// TwinCAT 3 PLC project ExtruderControl
// ProgramVersion: 3.1.4023.0
// libraries:
//   Tc2_ControllerToolbox, * (Beckhoff Automation GmbH)
//   Tc2_MC2, * (Beckhoff Automation GmbH)
//   Tc2_MC2_FlyingSaw, * (Beckhoff Automation GmbH)
//   Tc2_Standard, * (Beckhoff Automation GmbH)
//   Tc2_System, * (Beckhoff Automation GmbH)
//   Tc2_TempController, * (Beckhoff Automation GmbH)
//   Tc3_Database, * (Beckhoff Automation GmbH)
//   Tc3_Module, * (Beckhoff Automation GmbH)
//   VisuDialogs, * (System)
//   VisuSymbols,3.5.10.0,System
// project tree:
//   DUTs/ Modes.TcDUT, ST_CTRL_TempCtrlParameter2.TcDUT, ST_Material.TcDUT
//   DUTs/Vision/ PlcToSensor.TcDUT (not stored), SensorToPlc.TcDUT, VisionCmd.TcDUT, VisionState.TcDUT
//   / GlobalTextList.TcGTLO, PlcTask.TcTTO (not stored), Visualization Manager.TcVMO (not stored)
//   GVLs/ GVL.TcGVL, HMI.TcGVL, IO.TcGVL, MC.TcGVL
//   POUs/ AutoExtrusion.TcPOU (not stored), ControlTemp.TcPOU, GestionVentiladores.TcPOU, MedidaDiamMec.TcPOU, MedidaTempPuente.TcPOU, MAIN.TcPOU, MedidaTempTarjeta.TcPOU, Motion.TcPOU, OperatingModes.TcPOU
//   POUs/Database/ DatabaseManager.TcPOU
//   POUs/Operation/ Basic.TcPOU, Manual.TcPOU
//   POUs/Vision/ SensorFQM.TcPOU
//   POUs/VISUCode/ VisuLogic.TcPOU
//   VISUs/ BasicHMI.TcVIS, MainHMI.TcVIS, ManualHMI.TcVIS, VisionHMI.TcVIS
// real-time tasks:
//   TASK PlcTask: cycle T#10ms, priority 20, ADS port 350
// motion (NC):
//   TASK NC-Task Extruder SAF: cycle T#2ms, priority 4, ADS port 501
//   TASK NC-Task Extruder SVB: cycle T#10ms, priority 8, ADS port 511
//   AXIS ExtruderAxis (id 1)
//     Velo: FastManual=1300
//     PositionAreaControl: Range=50
//     OtherSettings: AllowMotionCmdToSlave=true
//     encoder EncType=8
//       EncPara: ScaleFactorNumerator=360, ScaleFactorDenominator=8388608, Inverse=true, MaxCount=#xffffffff
//     drive DrvType=9
//       DrvPara: Inverse=true, MaxCount=#xffffffff, DriveControlDWord=#x00030000
//         Analog: VeloScale=1.02398817080127, TorqueSetpointScale=10, ScaleFactorActTorque=0.1
//         TimeComp: TaskDelayCycles=1
//     controller CtrType=1
//       CtrPara: PriorControlFactor=1
//         PosDiffControl: Range=50
//         Observer: BandWidth=20
//   AXIS PullerAxis (id 2)
//     General: UnitName=Degree
//     Dynamic: Acceleration=68391, Deceleration=68391, Jerk=205173
//     Velo: RefSearch=455.94, RefSync=455.94, SlowManual=2279.7, FastManual=13678.2, Fast=45594, Maximum=45594
//     OtherSettings: AllowMotionCmdToSlave=true
//     encoder EncType=8
//       EncPara: ScaleFactorNumerator=360, ScaleFactorDenominator=1048576, MaxCount=#xffffffff
//     drive DrvType=9
//       DrvPara: MaxCount=#xffffffff, DriveControlDWord=#x00030000
//         Analog: VeloReferenz=50153.4, VeloScale=1.02398817080127, TorqueSetpointScale=10, ScaleFactorActTorque=0.1
//         TimeComp: TaskDelayCycles=1
//     controller CtrType=1
//       CtrPara: PriorControlFactor=1
//         Observer: BandWidth=20
//   AXIS PullerAxisVirtual (id 3)
//     General: UnitName=Degree
//     OtherSettings: AllowMotionCmdToSlave=true
//     encoder EncType=1
//       EncPara: ScaleFactorNumerator=1
//     drive DrvType=5
//       Analog: TorqueSetpointScale=10, ScaleFactorActTorque=0.1
//       TimeComp: TaskDelayCycles=1
//     controller CtrType=1
//       CtrPara: PriorControlFactor=1
//         Observer: BandWidth=20
// I/O:
//   DEVICE Dispositivo 2 (EtherCAT), AmsNetId 192.168.56.1.3.1
//     Term 1 (EK1100) [EK1100 EtherCAT Coupler (2A E-Bus)]
//       Term 2 (EL2008) [EL2008 8Ch. Dig. Output 24V, 0.5A]
//       Term 6 (EL3102) [EL3102 2Ch. Ana. Input +/-10V, Diff.]
//       Term 8 (EL3102) [EL3102 2Ch. Ana. Input +/-10V, Diff.]
//       Term 11 (EL3202) [EL3202 2Ch. Ana. Input PT100 (RTD)]
//       Term 13 (EL4132) [EL4132 2Ch. Ana. Output +/-10V]
//       Term 15 (EL9011) [EL9011 End Terminal]
//     Drive 3 (AX5206-0000-0011) [AX5206-0000-0011 EtherCAT Drive (SoE, 2 Ch.)]
//     Nº de boxes 7 (FQ-MS12x-ECT) [FQ-MS12x-ECT]
// variable links:
//   NC-Task Extruder SAF/Axes/ExtruderAxis <-> Device 2 (EtherCAT)/Drive 3 (AX5206-0000-0011)
//     Drive/Inputs/In/nDcOutputTime <-> InfoData/DcOutputShift
//     Drive/Inputs/In/nState1 <-> AT 1/Drive status word @bit 8
//     Drive/Inputs/In/nState2 <-> AT 1/Drive status word
//     Drive/Inputs/In/nState4 @bit 1 <-> WcState/InputToggle
//     Drive/Inputs/In/nState4 <-> WcState/WcState
//     Drive/Outputs/Out/nCtrl1 <-> MDT 1/Master control word @bit 8
//     Drive/Outputs/Out/nDataOut2 <-> MDT 1/Velocity command value
//     Enc/Inputs/In/nDataIn1 <-> AT 1/Position feedback 1 value
//     Enc/Inputs/In/nDcInputTime <-> InfoData/DcInputShift
//     Enc/Inputs/In/nState4 @bit 1 <-> WcState/InputToggle
//     Enc/Inputs/In/nState4 <-> WcState/WcState
//   NC-Task Extruder SAF/Axes/PullerAxis <-> Device 2 (EtherCAT)/Drive 3 (AX5206-0000-0011)
//     Drive/Inputs/In/nDcOutputTime <-> InfoData/DcOutputShift
//     Drive/Inputs/In/nState1 <-> AT 2/Drive status word @bit 8
//     Drive/Inputs/In/nState2 <-> AT 2/Drive status word
//     Drive/Inputs/In/nState4 @bit 1 <-> WcState/InputToggle
//     Drive/Inputs/In/nState4 <-> WcState/WcState
//     Drive/Outputs/Out/nCtrl1 <-> MDT 2/Master control word @bit 8
//     Drive/Outputs/Out/nDataOut2 <-> MDT 2/Velocity command value
//     Enc/Inputs/In/nDataIn1 <-> AT 2/Position feedback 1 value
//     Enc/Inputs/In/nDcInputTime <-> InfoData/DcInputShift
//     Enc/Inputs/In/nState4 @bit 1 <-> WcState/InputToggle
//     Enc/Inputs/In/nState4 <-> WcState/WcState
//   ExtruderControl/ExtruderControl Instance <-> Device 2 (EtherCAT)/Nº de boxes 7 (FQ-MS12x-ECT)
//     PlcTask Inputs/GVL.Vision.SensorToPlc/VisionDataOutput <-> 259th transmit PDO Mapping/Vision Data Output1
//     PlcTask Inputs/GVL.Vision.SensorToPlc/VisionDataOutput @bit {32..224 step 32} <-> 259th transmit PDO Mapping/Vision Data Output{2..8}  (7 links)
//     PlcTask Inputs/GVL.Vision.SensorToPlc/VisionResponseCode <-> 258th transmit PDO Mapping/Vision Response Code
//     PlcTask Inputs/GVL.Vision.SensorToPlc/VisionResponseData <-> 258th transmit PDO Mapping/Vision Response Data1
//     PlcTask Inputs/GVL.Vision.SensorToPlc/VisionStatusFlag @bit 1 <-> 257th transmit PDO Mapping/BUSY Bit
//     PlcTask Inputs/GVL.Vision.SensorToPlc/VisionStatusFlag @bit 15 <-> 257th transmit PDO Mapping/ERR Bit
//     PlcTask Inputs/GVL.Vision.SensorToPlc/VisionStatusFlag <-> 257th transmit PDO Mapping/FLG Bit
//     PlcTask Inputs/GVL.Vision.SensorToPlc/VisionStatusFlag @bit 16 <-> 257th transmit PDO Mapping/GATE Bit
//     PlcTask Inputs/GVL.Vision.SensorToPlc/VisionStatusFlag @bit 3 <-> 257th transmit PDO Mapping/OR Bit
//     PlcTask Inputs/GVL.Vision.SensorToPlc/VisionStatusFlag @bit 2 <-> 257th transmit PDO Mapping/READY Bit
//     PlcTask Inputs/GVL.Vision.SensorToPlc/VisionStatusFlag @bit 4 <-> 257th transmit PDO Mapping/RUN Bit
//     PlcTask Inputs/GVL.Vision.SensorToPlc/VisionStatusFlag @bit 5 <-> 257th transmit PDO Mapping/Status Reserve Bit05
//     PlcTask Inputs/GVL.Vision.SensorToPlc/VisionStatusFlag @bit 6 <-> 257th transmit PDO Mapping/Status Reserve Bit06
//     PlcTask Inputs/GVL.Vision.SensorToPlc/VisionStatusFlag @bit 7 <-> 257th transmit PDO Mapping/Status Reserve Bit07
//     PlcTask Inputs/GVL.Vision.SensorToPlc/VisionStatusFlag @bit 8 <-> 257th transmit PDO Mapping/Status Reserve Bit08
//     PlcTask Inputs/GVL.Vision.SensorToPlc/VisionStatusFlag @bit 9 <-> 257th transmit PDO Mapping/Status Reserve Bit09
//     PlcTask Inputs/GVL.Vision.SensorToPlc/VisionStatusFlag @bit 10 <-> 257th transmit PDO Mapping/Status Reserve Bit10
//     PlcTask Inputs/GVL.Vision.SensorToPlc/VisionStatusFlag @bit 11 <-> 257th transmit PDO Mapping/Status Reserve Bit11
//     PlcTask Inputs/GVL.Vision.SensorToPlc/VisionStatusFlag @bit 12 <-> 257th transmit PDO Mapping/Status Reserve Bit12
//     PlcTask Inputs/GVL.Vision.SensorToPlc/VisionStatusFlag @bit 13 <-> 257th transmit PDO Mapping/Status Reserve Bit13
//     PlcTask Inputs/GVL.Vision.SensorToPlc/VisionStatusFlag @bit 14 <-> 257th transmit PDO Mapping/Status Reserve Bit14
//     PlcTask Inputs/GVL.Vision.SensorToPlc/VisionStatusFlag @bit 17 <-> 257th transmit PDO Mapping/Status Reserve Bit17
//     PlcTask Inputs/GVL.Vision.SensorToPlc/VisionStatusFlag @bit 18 <-> 257th transmit PDO Mapping/Status Reserve Bit18
//     PlcTask Inputs/GVL.Vision.SensorToPlc/VisionStatusFlag @bit 19 <-> 257th transmit PDO Mapping/Status Reserve Bit19
//     PlcTask Inputs/GVL.Vision.SensorToPlc/VisionStatusFlag @bit 20 <-> 257th transmit PDO Mapping/Status Reserve Bit20
//     PlcTask Inputs/GVL.Vision.SensorToPlc/VisionStatusFlag @bit 21 <-> 257th transmit PDO Mapping/Status Reserve Bit21
//     PlcTask Inputs/GVL.Vision.SensorToPlc/VisionStatusFlag @bit 22 <-> 257th transmit PDO Mapping/Status Reserve Bit22
//     PlcTask Inputs/GVL.Vision.SensorToPlc/VisionStatusFlag @bit 23 <-> 257th transmit PDO Mapping/Status Reserve Bit23
//     PlcTask Inputs/GVL.Vision.SensorToPlc/VisionStatusFlag @bit 24 <-> 257th transmit PDO Mapping/Status Reserve Bit24
//     PlcTask Inputs/GVL.Vision.SensorToPlc/VisionStatusFlag @bit 25 <-> 257th transmit PDO Mapping/Status Reserve Bit25
//     PlcTask Inputs/GVL.Vision.SensorToPlc/VisionStatusFlag @bit 26 <-> 257th transmit PDO Mapping/Status Reserve Bit26
//     PlcTask Inputs/GVL.Vision.SensorToPlc/VisionStatusFlag @bit 27 <-> 257th transmit PDO Mapping/Status Reserve Bit27
//     PlcTask Inputs/GVL.Vision.SensorToPlc/VisionStatusFlag @bit 28 <-> 257th transmit PDO Mapping/Status Reserve Bit28
//     PlcTask Inputs/GVL.Vision.SensorToPlc/VisionStatusFlag @bit 29 <-> 257th transmit PDO Mapping/Status Reserve Bit29
//     PlcTask Inputs/GVL.Vision.SensorToPlc/VisionStatusFlag @bit 30 <-> 257th transmit PDO Mapping/Status Reserve Bit30
//     PlcTask Inputs/GVL.Vision.SensorToPlc/VisionStatusFlag @bit 31 <-> 257th transmit PDO Mapping/Status Reserve Bit31
//     PlcTask Outputs/GVL.Vision.PlcToSensor/VisionCommand <-> 258th receive PDO Mapping/Vision Command
//     PlcTask Outputs/GVL.Vision.PlcToSensor/VisionControlFlag @bit 2 <-> 257th receive PDO Mapping/Control Reserve Bit02
//     PlcTask Outputs/GVL.Vision.PlcToSensor/VisionControlFlag @bit 3 <-> 257th receive PDO Mapping/Control Reserve Bit03
//     PlcTask Outputs/GVL.Vision.PlcToSensor/VisionControlFlag @bit 4 <-> 257th receive PDO Mapping/Control Reserve Bit04
//     PlcTask Outputs/GVL.Vision.PlcToSensor/VisionControlFlag @bit 5 <-> 257th receive PDO Mapping/Control Reserve Bit05
//     PlcTask Outputs/GVL.Vision.PlcToSensor/VisionControlFlag @bit 6 <-> 257th receive PDO Mapping/Control Reserve Bit06
//     PlcTask Outputs/GVL.Vision.PlcToSensor/VisionControlFlag @bit 7 <-> 257th receive PDO Mapping/Control Reserve Bit07
//     PlcTask Outputs/GVL.Vision.PlcToSensor/VisionControlFlag @bit 8 <-> 257th receive PDO Mapping/Control Reserve Bit08
//     PlcTask Outputs/GVL.Vision.PlcToSensor/VisionControlFlag @bit 9 <-> 257th receive PDO Mapping/Control Reserve Bit09
//     PlcTask Outputs/GVL.Vision.PlcToSensor/VisionControlFlag @bit 10 <-> 257th receive PDO Mapping/Control Reserve Bit10
//     PlcTask Outputs/GVL.Vision.PlcToSensor/VisionControlFlag @bit 11 <-> 257th receive PDO Mapping/Control Reserve Bit11
//     PlcTask Outputs/GVL.Vision.PlcToSensor/VisionControlFlag @bit 12 <-> 257th receive PDO Mapping/Control Reserve Bit12
//     PlcTask Outputs/GVL.Vision.PlcToSensor/VisionControlFlag @bit 13 <-> 257th receive PDO Mapping/Control Reserve Bit13
//     PlcTask Outputs/GVL.Vision.PlcToSensor/VisionControlFlag @bit 14 <-> 257th receive PDO Mapping/Control Reserve Bit14
//     PlcTask Outputs/GVL.Vision.PlcToSensor/VisionControlFlag @bit 17 <-> 257th receive PDO Mapping/Control Reserve Bit17
//     PlcTask Outputs/GVL.Vision.PlcToSensor/VisionControlFlag @bit 18 <-> 257th receive PDO Mapping/Control Reserve Bit18
//     PlcTask Outputs/GVL.Vision.PlcToSensor/VisionControlFlag @bit 19 <-> 257th receive PDO Mapping/Control Reserve Bit19
//     PlcTask Outputs/GVL.Vision.PlcToSensor/VisionControlFlag @bit 20 <-> 257th receive PDO Mapping/Control Reserve Bit20
//     PlcTask Outputs/GVL.Vision.PlcToSensor/VisionControlFlag @bit 21 <-> 257th receive PDO Mapping/Control Reserve Bit21
//     PlcTask Outputs/GVL.Vision.PlcToSensor/VisionControlFlag @bit 22 <-> 257th receive PDO Mapping/Control Reserve Bit22
//     PlcTask Outputs/GVL.Vision.PlcToSensor/VisionControlFlag @bit 23 <-> 257th receive PDO Mapping/Control Reserve Bit23
//     PlcTask Outputs/GVL.Vision.PlcToSensor/VisionControlFlag @bit 24 <-> 257th receive PDO Mapping/Control Reserve Bit24
//     PlcTask Outputs/GVL.Vision.PlcToSensor/VisionControlFlag @bit 25 <-> 257th receive PDO Mapping/Control Reserve Bit25
//     PlcTask Outputs/GVL.Vision.PlcToSensor/VisionControlFlag @bit 26 <-> 257th receive PDO Mapping/Control Reserve Bit26
//     PlcTask Outputs/GVL.Vision.PlcToSensor/VisionControlFlag @bit 27 <-> 257th receive PDO Mapping/Control Reserve Bit27
//     PlcTask Outputs/GVL.Vision.PlcToSensor/VisionControlFlag @bit 28 <-> 257th receive PDO Mapping/Control Reserve Bit28
//     PlcTask Outputs/GVL.Vision.PlcToSensor/VisionControlFlag @bit 29 <-> 257th receive PDO Mapping/Control Reserve Bit29
//     PlcTask Outputs/GVL.Vision.PlcToSensor/VisionControlFlag @bit 30 <-> 257th receive PDO Mapping/Control Reserve Bit30
//     PlcTask Outputs/GVL.Vision.PlcToSensor/VisionControlFlag @bit 31 <-> 257th receive PDO Mapping/Control Reserve Bit31
//     PlcTask Outputs/GVL.Vision.PlcToSensor/VisionControlFlag @bit 16 <-> 257th receive PDO Mapping/DSA Bit
//     PlcTask Outputs/GVL.Vision.PlcToSensor/VisionControlFlag @bit 15 <-> 257th receive PDO Mapping/ERCLR Bit
//     PlcTask Outputs/GVL.Vision.PlcToSensor/VisionControlFlag <-> 257th receive PDO Mapping/EXE Bit
//     PlcTask Outputs/GVL.Vision.PlcToSensor/VisionControlFlag @bit 1 <-> 257th receive PDO Mapping/TRIG Bit
//   ExtruderControl/ExtruderControl Instance <-> Device 2 (EtherCAT)/Term 1 (EK1100)/Term 11 (EL3202)
//     PlcTask Inputs/IO.I_TermB <-> RTD Inputs Channel 2/Value
//     PlcTask Inputs/IO.I_TermT <-> RTD Inputs Channel 1/Value
//   ExtruderControl/ExtruderControl Instance <-> Device 2 (EtherCAT)/Term 1 (EK1100)/Term 13 (EL4132)
//     PlcTask Outputs/IO.Q_Vent1 <-> Channel 1/Output
//     PlcTask Outputs/IO.Q_Vent2 <-> Channel 2/Output
//   ExtruderControl/ExtruderControl Instance <-> Device 2 (EtherCAT)/Term 1 (EK1100)/Term 2 (EL2008)
//     PlcTask Outputs/IO.Q_HeaterB <-> Channel 2/Output
//     PlcTask Outputs/IO.Q_HeaterT <-> Channel 1/Output
//     PlcTask Outputs/IO.Q_VisionLight <-> Channel 3/Output
//   ExtruderControl/ExtruderControl Instance <-> Device 2 (EtherCAT)/Term 1 (EK1100)/Term 6 (EL3102)
//     PlcTask Inputs/IO.I_SMec1 <-> Channel 1/Value
//     PlcTask Inputs/IO.I_SMec2 <-> Channel 2/Value
//   ExtruderControl/ExtruderControl Instance <-> Device 2 (EtherCAT)/Term 1 (EK1100)/Term 8 (EL3102)
//     PlcTask Inputs/IO.I_TermBPuente <-> Channel 2/Value
//     PlcTask Inputs/IO.I_TermTPuente <-> Channel 1/Value
//   ExtruderControl/ExtruderControl Instance <-> NC-Task Extruder SAF/Axes/ExtruderAxis
//     PlcTask Inputs/MC.Extruder.NcToPlc <-> Outputs/ToPlc
//     PlcTask Outputs/MC.Extruder.PlcToNc <-> Inputs/FromPlc
//   ExtruderControl/ExtruderControl Instance <-> NC-Task Extruder SAF/Axes/PullerAxis
//     PlcTask Inputs/MC.Puller.NcToPlc <-> Outputs/ToPlc
//     PlcTask Outputs/MC.Puller.PlcToNc <-> Inputs/FromPlc
//   ExtruderControl/ExtruderControl Instance <-> NC-Task Extruder SAF/Axes/PullerAxisVirtual
//     PlcTask Inputs/MC.PullerVirtual.NcToPlc <-> Outputs/ToPlc
//     PlcTask Outputs/MC.PullerVirtual.PlcToNc <-> Inputs/FromPlc

// ---- DUTs/Modes.TcDUT
{attribute 'qualified_only'}
{attribute 'strict'}
TYPE Modes :
(
	STOP_EM := 0,
	STOP_OP := 1,
	AUTO := 2,
	MAN := 3,
	Stopping := 4
);
END_TYPE

// ---- DUTs/ST_CTRL_TempCtrlParameter2.TcDUT
TYPE ST_CTRL_TempCtrlParameter2 :
STRUCT
  (* general parameters *)
  iMode                     : E_CTRL_ControlMode:=1;
  iReactionOnFailure        : E_CTRL_ReactionOnFailure;
  bSelCtrlParameterSet      : BOOL:=FALSE;
  dwAlarmSupp               : DWORD;
  tCtrlCycleTime            : TIME:=T#100MS;
  tTaskCycleTime            : TIME:=T#10MS;

  (* tuning parameteer *)
  iTuningMode               : E_CTRL_TuneMode:= eCTRL_TuneMode_heating;
  tTuneStabilisation        : TIME       := T#20S;
  fEndTunePercentHeating    : LREAL      := 80.0;
  fYTuneHeating             : LREAL;
  fYStableHeating           : LREAL;
  fEndTunePercentCooling    : LREAL      := 20.0;
  fYTuneCooling             : LREAL;
  fYStableCooling           : LREAL;
  fScalingFactor            : LREAL      := 1.0;

  (* setpoint parameters *)
  fWMin                     : LREAL;
  fWMax                     : LREAL;

  (* start up *)
  bEnableSoftStart          : BOOL;
  bEnableRamping            : BOOL;
  fWStartUp                 : LREAL;
  tStartUp                  : TIME;
  bStartUpRamping           : BOOL;
  fWStartUpVeloPos          : LREAL;
  fWStartUpVeloNeg          : LREAL;
  fWVeloPos                 : LREAL;
  fWVeloNeg                 : LREAL;

  (* actual value parameters *)
  bFilter                   : BOOL;
  tFilter                   : TIME;

  (* deadband parameters *)
  bDeadband                 : BOOL;
  fEDeadband                : LREAL;
  
  (* control value parameters *)
  fYMin                     : LREAL;
  fYMax                     : LREAL;
  fYManual                  : LREAL;
  fYOnFailure               : LREAL;
  tPWMCycleTime             : TIME;
  tPWMMinOffTime            : TIME;
  tPWMMinOnTime             : TIME;
  tPWMWaitingTime           : TIME;
  fYThresholdOff            : LREAL;
  fYThresholdOn             : LREAL;
  nCyclesForSwitchOver      : INT        := 100;

  (* controller settings *)
  bEnablePreController      : BOOL;
  bEnableZones              : BOOL;
  bEnableCVFilter           : BOOL;
  iFilterType               : E_CTRL_FilterType;
  iControllerType           : E_CTRL_ControllerType;

  (* min max temperatures *)
  TempLow                   : LREAL;
  TempLowLow                : LREAL;
  TempHigh                  : LREAL;
  TempHighHigh              : LREAL;
  TempAbsoluteHigh          : LREAL;
  TempAbsoluteLow           : LREAL;

  (* internal tuning parameters *)
  fTuneKp                   : LREAL     := 1.2;
  fTuneTn                   : LREAL     := 2.0;
  fTuneTv                   : LREAL     := 0.42;
  fTuneTd                   : LREAL     := 0.25;
END_STRUCT
END_TYPE

// ---- DUTs/ST_Material.TcDUT
TYPE ST_Material :
STRUCT
	ID: ARRAY[0..15] OF BYTE;
	Name: STRING(50);
	Description: STRING(255);
	BedTemperature: LREAL;
	HotendTemperature: LREAL;
	IdealTempExtr: LREAL;
	MinTempExtr: LREAL;
	MaxTempExtr: LREAL;
END_STRUCT
END_TYPE

// ---- DUTs/Vision/SensorToPlc.TcDUT
TYPE SensorToPlc :
STRUCT
	VisionStatusFlag AT %I*:DWORD; //Doble Palabra que contiene los bits siguientes
	FLG:BOOL; //Posicion 0
	BUSY:BOOL; //Posicion 1
	READY:BOOL; //Posicion 2
	OR_Jud:BOOL; //Posicion 3
	RUN:BOOL; //Posicion 4
	ERR:BOOL; //Posicion 15
	GATE:BOOL; //Posicion 16
	
	VisionResponseCode AT %I*:DWORD;
	VisionResponseData AT %I*:DWORD;
	
	//Lecturas desde el sensor
	VisionDataOutput AT %I*: ARRAY [0..7] OF REAL;
END_STRUCT
END_TYPE

// ---- DUTs/Vision/VisionCmd.TcDUT
{attribute 'qualified_only'}
{attribute 'strict'}
TYPE VisionCmd :
(
	StartSingle := 0,
	StartContinuous := 1,
	StopContinuous := 2,
	ClearValues := 3,
	ClearDataOutputBuffer := 4,
	Reset := 5,
	GetLatestError := 6
);
END_TYPE;

// ---- DUTs/Vision/VisionState.TcDUT
{attribute 'qualified_only'}
{attribute 'strict'}
TYPE VisionState :
(
	Error := 000,
	Checking_error := 001,
	Clear_data := 002,
	Clear_error := 003,
	StandStill := 010,
	Switching_Single := 011,
	Switching_Continuous := 012,
	ContinuousMeasurement := 020,
	Stopping_Continuous := 021,
	SingleMeasurement := 030,
	TakingSingleMeasurement := 031,
	EmptyDebug := 999
);
END_TYPE

// ---- GVLs/GVL.TcGVL
{attribute 'qualified_only'}
VAR_GLOBAL
	
	Mode: Modes;
	Vision:SensorFQM;
	VisionResults:ARRAY [0..7] OF REAL;
	VisionResultsmm:ARRAY [0..7] OF REAL;
	//ScalingFactor:REAL:= 0.0414;
	ScalingFactor:REAL:= 0.03798; 	//Factor de escalado (mm/pixeles) para broca de 1.75mm
	
	NuevaMedidaCamara:BOOL:=FALSE; 	//Variable auxiliar para el control de la camara
	
	//Variables para el control de la temperatura
	TempTerT: LREAL; 	//Temperatura medida por el Pt100 del termico superior
	TempTerB: LREAL; 	//Temperatura medida por el Pt100 del termico inferior
	//TempExtrusion:REAL:=205;	//Temperatura de extrusion dependiendo del material (PLA)
	TempExtrusion:REAL:=195;	//Para pruebas
	
	//Variables para el control del diametro del filamento con el sensor mecanico
	MedidaSensorMecanico:REAL:=0.0;		//Media de medidas y por tanto medida del diametro
	
	//Variables para el control del diametro
	config:BOOL:=0; 			//0 para 1.75mm y 1 para 2.85mm de diametro
	dReferencia:REAL:=1.75; 	//1.75 o 2.85
	//Estos valores (vPaso y dTolerancia) habría que asignarlos de forma correcta segun los parametros del motor inferior
	vPaso:INT:=2; 				//Valor para variar la velocidad de actuacion de los rodillos inferiores
	dTolerancia:REAL:=0.03; 	//Tolerancia permitida en la medida del diametro del filamento
	
	//Variable para controlar velocidad del motor inferior (puller)
	//A estas variables habria que asignarle unos valores correctos para realizar el control de forma optima
	ActPuller: LREAL; 			//Valor inicial de actuacion que variara segun el valor del diametro
	ActPuller_Max: LREAL;
	ActPuller_Min: LREAL;
	
	State:INT:= 0; //Para gestion de la maquina de estados
	//0: estado inicial
	//1: dar potencia
	//2: calentar 
	//3: mover en velocidad extrusora y puller
	//4: funcionamiento extrusora
	//5: nueva foto y gestion de termicos
	//6: calculo de la nueva velocidad
	//7: cambio de velocidad del puller
	//30: parar ejes
END_VAR

// ---- GVLs/HMI.TcGVL
{attribute 'qualified_only'}
VAR_GLOBAL
	
	// Modes control
	Bt_Run: BOOL;
	Bt_Stop: BOOL;
	S_ManAuto: BOOL := TRUE;
	Bt_EmStop: BOOL;
	Bt_Rearm:BOOL;
	Bt_Front: BOOL;
	Bt_Back:BOOL;
	
	//Process Control
	Bt_StartCycle:BOOL;
	Bt_StopCycle:BOOL;
	Bt_ResetAxis:BOOL;
	Tb_Vel:LREAL;
	Tb_TempB:LREAL;
	Tb_TempT:LREAL;
	Tb_Temp:LREAL;
	
	//Vision control
	Bt_ActivateContinuous:BOOL;
	Bt_ActivateSingle:BOOL;
	Bt_Shot:BOOL;
	L_NewMeasurement:BOOL;
	
	//Manual HMI
	Bt_ManHeatTop:BOOL;
	Bt_ManHeatBot:BOOL;
	Bt_ManForwardExtruder:BOOL;
	Bt_ManBackwardsExtruder:BOOL;
	Bt_Light:BOOL;
	Tb_ManVelExtruder:REAL;
	Bt_ManForwardPuller:BOOL;
	Bt_ManBackwardsPuller:BOOL;
	Tb_ManVelPuller:REAL;
	
END_VAR

VAR_GLOBAL CONSTANT
	MeasurementNames: ARRAY [0..7] OF STRING:= ['Top diameter','Mid diameter','Low diameter','Empty','Empty','Empty','Empty','Empty'];
END_VAR

// ---- GVLs/IO.TcGVL
{attribute 'qualified_only'}
VAR_GLOBAL
	
	// Heater outputs
	Q_HeaterT AT %Q*:BOOL;
	Q_HeaterB AT %Q*:BOOL;
	Q_VisionLight AT %Q*:BOOL;
	
	// RTD Sensors (PT100)
	I_TermT AT %I*:INT;
	I_TermB AT %I*:INT;
	
	// Valor temperatura puente de resistencias
	I_TermTPuente AT %I*:INT;
	I_TermBPuente AT %I*:INT;
	
	// Sensores mecanicos diametro
	I_SMec1 AT %I*:INT;
	I_SMec2 AT %I*:INT;
	
	//Ventiladores
	Q_Vent1 AT %Q*:INT;
	Q_Vent2 AT %Q*:INT;
	
END_VAR

// ---- GVLs/MC.TcGVL
{attribute 'qualified_only'}
VAR_GLOBAL
	// Axis ref
	Extruder: AXIS_REF;
	Puller: AXIS_REF;
	PullerVirtual:AXIS_REF; //Eje virtual para controlar el Puller
	
	// Orders
	En_Power:BOOL;
	Exec_Stop:BOOL;
	Exec_Velocity:BOOL;
	Exec_Relative:BOOL;
	Exec_Reset:BOOL;
	
	Man_ForwardExtruder:BOOL;
	Man_BackwardsExtruder:BOOL;
	
	Man_ForwardPuller:BOOL;
	Man_BackwardsPuller:BOOL;
	
	// Motion variables
	Override:LREAL := 100;
	TargetVel:LREAL;
	TargetPosRel:LREAL;
	TargetDirection:MC_Direction;
	
	// Puller
	PullerVel:LREAL;
	Exec_VelocityPuller:BOOL;
	PullerDirection:MC_Direction;
	Acoplar:BOOL;
	Desacoplar:BOOL;
END_VAR

VAR_GLOBAL CONSTANT
	// Motion constants
	StdVel:LREAL:= 100;
	StdAcc:LREAL:= 1000;
	StdDecc:LREAL:= 1000;
END_VAR

// ---- POUs/Vision/SensorFQM.TcPOU
FUNCTION_BLOCK SensorFQM
VAR_INPUT
END_VAR
VAR_OUTPUT
END_VAR
VAR_IN_OUT
	
END_VAR
VAR
	State:VisionState:= 0;
	SensorToPlc AT %I*:SensorToPlc;
	PlcToSensor AT %Q*:PlcToSensor;
	KeepAliveTimer:TON;
	
	RExec:R_TRIG;
	NextCycleResetFlags:BOOL;
	Results: ARRAY [0..7] OF REAL;
	
	//Single measurement
	RequestSingle:BOOL;
	TakePhoto:BOOL;
	TakePhotoFlag:R_TRIG;
	MeasureTimer:TON;
	MeasureTime:TIME;
	
	//Continuous measurement
	RequestStartCont:BOOL;
	RequestStopCont:BOOL;
	StopFromError:BOOL;
	ResponseTimer:TON;
	ResponseTime:TIME;
	FEnable:F_TRIG;
	
	LastResult:INT:=0;//0-Null, 1-Ok, 2-NG
	
	//Error Management
	RequestErrorCode:BOOL;
	LastError:DWORD;
END_VAR
VAR CONSTANT
	KeepAliveBit:INT:=24;
END_VAR

// Preparing Inputs
SensorToPlc.FLG:= SensorToPlc.VisionStatusFlag.0;
SensorToPlc.BUSY:= SensorToPlc.VisionStatusFlag.1;
SensorToPlc.READY:= SensorToPlc.VisionStatusFlag.2;
SensorToPlc.OR_Jud:= SensorToPlc.VisionStatusFlag.3;
SensorToPlc.RUN:= SensorToPlc.VisionStatusFlag.4;
SensorToPlc.ERR:= SensorToPlc.VisionStatusFlag.15;
SensorToPlc.GATE:= SensorToPlc.VisionStatusFlag.16;
//Change a bit every 500ms as Keep Alive bit
(*KeepAliveTimer(in:=NOT KeepAliveTimer.Q, pt:=T#1S);
IF KeepAliveTimer.Q THEN
	PlcToSensor.VisionControlFlag.24:= NOT PlcToSensor.VisionControlFlag.24;
END_IF*)

//Delete variables. Estado distinto de 999 para permitir modificar a mano en ese estado especial
IF State <> 999 THEN
	PlcToSensor.EXE:=FALSE;
	PlcToSensor.ERCLR:=FALSE;
	PlcToSensor.DSA:=FALSE;
	PlcToSensor.TRIG:=FALSE;
END_IF

//State machine
CASE State OF
	000: //Error. Por ahora se salta parada cuando hay error
		IF NOT SensorToPlc.ERR THEN
			State := 010;
		ELSE
			State := 001;
		END_IF
			
	001: //Checking errors
		//TODO: Revisar
		_prepareCommand(Command:= VisionCmd.GetLatestError);
		PlcToSensor.EXE := TRUE;
		IF SensorToPlc.FLG THEN
			PlcToSensor.EXE := FALSE;
			LastError:= SensorToPlc.VisionResponseData;
			State := 002;
		END_IF
	002: //Clear data
		_prepareCommand(VisionCmd.ClearDataOutputBuffer);
		PlcToSensor.EXE := TRUE;
		IF SensorToPlc.FLG THEN
			PlcToSensor.EXE := FALSE;
			State := 003;
		END_IF
	003: //Clear Error
		PlcToSensor.ERCLR:=TRUE;
		IF NOT SensorToPlc.ERR THEN
			PlcToSensor.ERCLR := FALSE;
			State := 010;
		END_IF
	010: //StandStill
		IF RequestSingle THEN
			LastError := 0; //Elimina ultimo error cuando se pasa a este estado
			State := 011;
		END_IF
		IF RequestStartCont AND NOT RequestSingle THEN
			State := 012;
		END_IF
		IF SensorToPlc.ERR THEN
			State := 001;
			
		END_IF
	011: //Switching to Single
		_prepareCommand(VisionCmd.StartSingle);
		PlcToSensor.EXE:=TRUE;
		IF SensorToPlc.FLG THEN
			PlcToSensor.EXE := FALSE;
			State := 030;
			LastResult:=0;
		END_IF
	012: //Switching to continuous
		_prepareCommand(VisionCmd.StartContinuous);
		PlcToSensor.EXE:=TRUE;
		IF SensorToPlc.FLG THEN
			PlcToSensor.EXE := FALSE;
			State := 020;
		END_IF
	020: //Continuous Measurement
		//Loop to request measurement
		IF SensorToPlc.GATE THEN
			ResponseTime:=ResponseTimer.ET;
			PlcToSensor.DSA := FALSE;
			ResponseTimer(in:=FALSE, pt:=T#10S);
		ELSIF NOT SensorToPLC.gate THEN
			ResponseTimer(in:=TRUE, pt:=T#10S);
			PlcToSensor.DSA := TRUE;
		END_IF
		//transitions
		IF SensorToPLC.ERR THEN
			PlcToSensor.EXE := FALSE;
			StopFromError:=TRUE;
			State := 021;
		END_IF 
		IF RequestStopCont THEN
			PlcToSensor.EXE := FALSE;
			State := 021;
		END_IF
	021: //Stopping continuous
	    _prepareCommand(VisionCmd.StopContinuous);
		PlcToSensor.EXE := TRUE;
		IF SensorToPLC.FLG THEN
			IF StopFromError THEN
				PlcToSensor.EXE :=FALSE;
				StopFromError:=FALSE;
				State := 001;
			ELSE
				State := 010;
			END_IF
			RequestStopCont := FALSE;
		END_IF
	030: // Single Measurement Ready
		
		IF TakePhoto THEN
			//Take photo and request
			PlcToSensor.TRIG:=TRUE;
			PlcToSensor.DSA:=TRUE;
			MeasureTimer(in:=FALSE);
			MeasureTimer(in:=TRUE, pt:=T#60s);
			State := 31;
		END_IF
		IF NOT RequestSingle THEN
			State := 010;
		END_IF
		IF SensorToPlc.ERR THEN
			State := 001;
			_prepareCommand(Command:= VisionCmd.GetLatestError);
			PlcToSensor.EXE := TRUE;
		END_IF
	031: // Single Measurement Taking photo
		PlcToSensor.DSA := TRUE; // Ojo, ya se activo en el ciclo anterior. no hay retardo de un ciclo.
		PlcToSensor.TRIG := TRUE;
		MeasureTimer(in:=TRUE);
		IF SensorToPLC.GATE THEN
			//TODO: Esto llega mas tarde que el dato. Revisar.
			IF SensorToPlc.OR_Jud THEN
				LastResult:=2;
			ELSE
				LastResult:=1;
			END_IF
			MeasureTime:=MeasureTimer.ET;
			MeasureTimer(in:=FALSE);
			State := 030;
			PlcToSensor.TRIG:=FALSE;
			PlcToSensor.DSA:=FALSE;
		END_IF
		IF SensorToPLC.ERR THEN
			State := 001;
		END_IF
END_CASE

//Update Flag Bits into DWORD
PlcToSensor.VisionControlFlag.0:= PlcToSensor.EXE;
PlcToSensor.VisionControlFlag.1:= PlcToSensor.TRIG;
PlcToSensor.VisionControlFlag.15:= PlcToSensor.ERCLR;
PlcToSensor.VisionControlFlag.16:= PlcToSensor.DSA;

METHOD PRIVATE _prepareCommand
VAR_INPUT
	Command:VisionCmd;
END_VAR
VAR
	
END_VAR
(* 
Command orders deliverable to camera.
See OMRON FQ-M Series Vision Sensor docs for information
*)
CASE Command OF
	VisionCmd.StartSingle: 				PlcToSensor.VisionCommand:= 16#00101010;
	VisionCmd.StartContinuous: 			PlcToSensor.VisionCommand:= 16#00101020;
	VisionCmd.StopContinuous: 			PlcToSensor.VisionCommand:= 16#00101030;
	VisionCmd.ClearValues: 				PlcToSensor.VisionCommand:= 16#00102010;
	VisionCmd.ClearDataOutputBuffer: 	PlcToSensor.VisionCommand:= 16#00102020;
	VisionCmd.Reset: 					PlcToSensor.VisionCommand:= 16#0010F010;
	VisionCmd.GetLatestError: 			PlcToSensor.VisionCommand:= 16#00205000;
END_CASE
END_METHOD

METHOD PUBLIC ContinuousShot : BOOL
VAR_INPUT
	Enable:BOOL; //Habilita el modo continuo. NOTA: Tendrá prioridad el modo único
END_VAR
VAR_OUTPUT
	Q:ARRAY [0..7] OF REAL;
END_VAR
FEnable(CLK:=Enable);
IF Enable THEN
	RequestStartCont:=TRUE;
	RequestStopCont:=FALSE;
END_IF
IF FEnable.Q THEN
	RequestStartCont:=FALSE;
	RequestStopCont:=TRUE;
	PlcToSensor.DSA:=FALSE;
	ResponseTimer(in:=FALSE);
END_IF

IF Enable THEN
//	IF SensorToPlc.GATE THEN
//		ResponseTime:=ResponseTimer.ET;
//		PlcToSensor.DSA := FALSE;
//		ResponseTimer(in:=FALSE, pt:=T#10S);
//	ELSIF NOT SensorToPLC.gate THEN
//		ResponseTimer(in:=TRUE, pt:=T#10S);
//		PlcToSensor.DSA := TRUE;
//	END_IF
;
END_IF

Q := SensorToPlc.VisionDataOutput;
END_METHOD

METHOD PUBLIC SingleShot : BOOL
VAR_INPUT
	Enable:BOOL;
	Execute:BOOL;
END_VAR
VAR_OUTPUT
	Active:BOOL;
	Measurement:BOOL;
	Ok:BOOL;
	Ng:BOOL;
	Q: ARRAY [0..7] OF REAL;
END_VAR
IF Enable THEN
	RequestSingle:=TRUE;
ELSE
	RequestSingle:=FALSE;
END_IF

TakePhotoFlag(clk:= Execute);
IF State = 030 THEN
	Active:=TRUE;
	IF TakePhotoFlag.Q THEN
		TakePhoto:=TRUE;
		Ok:=FALSE;
		Ng:=FALSE;
	END_IF
	CASE LastResult OF
		0: Ok:=FALSE; Ng:=FALSE; Measurement:=FALSE;
		1: Ok:=TRUE; Ng:=FALSE; Measurement:=TRUE;
		2: Ok:=FALSE; Ng:=TRUE; Measurement:= TRUE;
	END_CASE
	
ELSIF State = 031 THEN
	TakePhoto:=FALSE;
END_IF

Q := SensorToPlc.VisionDataOutput;
END_METHOD

END_FUNCTION_BLOCK

// ---- POUs/Operation/Manual.TcPOU
PROGRAM Manual
VAR
	
	ExitManual:F_TRIG;
	
	LoopCounter:INT;
	
	//Variables para la lectura de sensores
	MedSensores:REAL:=0.0;
	SumSenOpt: REAL:=0.0;
	MedSenOpt: REAL:=0.0;
	
	//Variables para la media de medidas de los sensores
	Lecturas:ARRAY[0..9] OF REAL:=[10(0.0)]; 	//Medidas del diametro inicializadas
	Index:INT:=0; 								//Indice del vector de medidas 
	Suma:REAL:=0.0; 							//Suma de medidas
	Medida:REAL:=0.0; 							//Media de medidas y por tanto medida del diametro
	
END_VAR

IF GVL.Mode = Modes.MAN THEN
	//Gestion de temperatura para extrusion.
	//IO.Q_HeaterB:=HMI.Bt_ManHeatBot;
	//IO.Q_HeaterT:=HMI.Bt_ManHeatTop;
	
	IF (GVL.TempTerT>(GVL.TempExtrusion*0.95)) OR (NOT HMI.Bt_ManHeatTop) THEN 	//Gestiona el calentador superior
		IO.Q_HeaterT:=FALSE;
	END_IF
	IF (GVL.TempTerT<(GVL.TempExtrusion*0.95-1.0)) AND HMI.Bt_ManHeatTop THEN
		IO.Q_HeaterT:=TRUE;
	END_IF
	
	IF (GVL.TempTerB>(GVL.TempExtrusion)) OR (NOT HMI.Bt_ManHeatBot) THEN 		//Gestiona el calentador inferior
		IO.Q_HeaterB:=FALSE;
	END_IF
	IF (GVL.TempTerB<(GVL.TempExtrusion-1.0))AND HMI.Bt_ManHeatBot THEN
		IO.Q_HeaterB:=TRUE;
	END_IF
	
	//Al pulsar botones, primero dar orden de potencia
	IF HMI.Bt_ManForwardExtruder OR HMI.Bt_ManBackwardsExtruder OR HMI.Bt_ManBackwardsPuller OR HMI.Bt_ManForwardPuller THEN
		MC.En_Power := TRUE;
		//Ya en potencia, se ejecuta la orden
		IF Motion.FB_Power.Status AND Motion.FB_Power2.Status AND Motion.FB_Power3.Status THEN
			MC.Man_ForwardExtruder := HMI.Bt_ManForwardExtruder;
			MC.Man_BackwardsExtruder := HMI.Bt_ManBackwardsExtruder;
			MC.Man_ForwardPuller:=HMI.Bt_ManForwardPuller;
			MC.Man_BackwardsPuller:=HMI.Bt_ManBackwardsPuller;
		END_IF
	//Si se deja de pulsar, al acabar movimiento, se quita potencia
	ELSE
		MC.Man_ForwardExtruder := FALSE;
		MC.Man_BackwardsExtruder := FALSE;
		MC.Man_ForwardPuller:=FALSE;
		MC.Man_BackwardsPuller:=FALSE;
		IF NOT Motion.FB_ManualExtruder.Busy AND NOT Motion.FB_ManualPuller.Busy THEN
			MC.En_Power := FALSE;
		ELSE
			MC.En_Power := TRUE;
		END_IF
	END_IF
//	MC.Man_Forward := HMI.Bt_ManForward;
//	MC.Man_Backwards := HMI.Bt_ManBackwards;
	IO.Q_VisionLight := HMI.Bt_Light;
	
	GVL.Vision.SingleShot(Enable:=HMI.Bt_ActivateSingle, 
						Execute:=HMI.Bt_Shot,
						Q=>GVL.VisionResults,
						Measurement=>GVL.NuevaMedidaCamara);
    GVL.Vision.ContinuousShot(Enable:=HMI.Bt_ActivateContinuous,
						Q=>GVL.VisionResults);		
	
	IF HMI.Bt_ActivateSingle AND GVL.NuevaMedidaCamara THEN
		// Restablecer valores de medida para una futura medida
		GVL.NuevaMedidaCamara:=FALSE;
		GVL.Vision.SingleShot(Enable:=TRUE, Execute:=FALSE);
		SumSenOpt:=0.0;
		FOR LoopCounter:=0 TO 7 BY 1 DO
			GVL.VisionResultsmm[LoopCounter] := GVL.VisionResults[LoopCounter]*GVL.ScalingFactor;
			SumSenOpt:=GVL.VisionResultsmm[LoopCounter]+SumSenOpt;
		END_FOR	
		MedSenOpt:=SumSenOpt/3;
		
		//Calculo del diametro
		MedSensores:=((GVL.MedidaSensorMecanico+MedSenOpt)/2);
		(*
		//Hacer media de las 10 ultimas medidas del diametro
		Suma:= Suma - Lecturas[Index];
		Lecturas[index]:=MedSensores;
		Suma:=Suma+Lecturas[index];
		Index:= Index + 1;
		IF (Index > 9) THEN
			Index := 0;    	//Volvemos al inicio del vector
		END_IF
		Medida:=Suma/10;
		*)
		(*
		//Gestion de la actuacion
		IF (MedSensores>(GVL.dReferencia+GVL.dTolerancia)) THEN 		//Diametro grande
			GVL.ActPuller:=GVL.ActPuller+GVL.vPaso;
		END_IF
	
		IF (MedSensores<(GVL.dReferencia-GVL.dTolerancia)) THEN 		//Diametro pequeño
			GVL.ActPuller:=GVL.ActPuller-GVL.vPaso;
		END_IF
	
		//Limitador de la actuacion
		IF (GVL.ActPuller>GVL.ActPuller_Max) THEN 
			GVL.ActPuller:=GVL.ActPuller_Max;
		ELSIF (GVL.ActPuller<GVL.ActPuller_Min) THEN
			GVL.ActPuller:=GVL.ActPuller_Min;
		END_IF
		*)
	END_IF
	IF HMI.Bt_ActivateContinuous THEN
		// Restablecer valores de medida para una futura medida
		SumSenOpt:=0.0;
		FOR LoopCounter:=0 TO 7 BY 1 DO
			GVL.VisionResultsmm[LoopCounter] := GVL.VisionResults[LoopCounter]*GVL.ScalingFactor;
			SumSenOpt:=GVL.VisionResultsmm[LoopCounter]+SumSenOpt;
		END_FOR	
		MedSenOpt:=SumSenOpt/3;
		
		//Calculo del diametro
		MedSensores:=((GVL.MedidaSensorMecanico+MedSenOpt)/2);
		
		//Hacer media de las 10 ultimas medidas del diametro
		Suma:= Suma - Lecturas[Index];
		Lecturas[index]:=MedSensores;
		Suma:=Suma+Lecturas[index];
		Index:= Index + 1;
		IF (Index > 9) THEN
			Index := 0;    	//Volvemos al inicio del vector
		END_IF
		Medida:=Suma/10;
		(*
		//Gestion de la actuacion
		IF (MedSensores>(GVL.dReferencia+GVL.dTolerancia)) THEN 		//Diametro grande
			GVL.ActPuller:=GVL.ActPuller+GVL.vPaso;
		END_IF
	
		IF (MedSensores<(GVL.dReferencia-GVL.dTolerancia)) THEN 		//Diametro pequeño
			GVL.ActPuller:=GVL.ActPuller-GVL.vPaso;
		END_IF
	
		//Limitador de la actuacion
		IF (GVL.ActPuller>GVL.ActPuller_Max) THEN 
			GVL.ActPuller:=GVL.ActPuller_Max;
		ELSIF (GVL.ActPuller<GVL.ActPuller_Min) THEN
			GVL.ActPuller:=GVL.ActPuller_Min;
		END_IF
		*)
	END_IF
	
ELSE
	HMI.Bt_ManHeatBot := FALSE;
	HMI.Bt_ManHeatTop:= FALSE;
	MC.Man_ForwardExtruder := FALSE;
	HMI.Bt_ManForwardExtruder := FALSE;
	MC.Man_BackwardsExtruder := FALSE;
	HMI.Bt_ManBackwardsExtruder := FALSE;
	MC.Man_ForwardPuller := FALSE;
	HMI.Bt_ManForwardPuller := FALSE;
	MC.Man_BackwardsPuller := FALSE;
	HMI.Bt_ManBackwardsPuller := FALSE;
	HMI.Bt_Light := FALSE;
	HMI.Bt_ActivateSingle:=FALSE;
	HMI.Bt_ActivateContinuous:=FALSE;
END_IF

ExitManual(clk:=(GVL.Mode = Modes.MAN));
IF ExitManual.Q THEN
	IO.Q_HeaterB := FALSE;
	IO.Q_HeaterT :=FALSE;
	IO.Q_VisionLight := FALSE;
END_IF

END_PROGRAM

// ---- POUs/Motion.TcPOU
PROGRAM Motion
VAR
	FB_Power: MC_Power;
	FB_Stop: MC_Stop;
	FB_StopPuller: MC_Stop;
	FB_StopPullerVirtual: MC_Stop;
	FB_Velocity: MC_MoveVelocity;
	FB_VelocityPuller: MC_MoveVelocity;
	FB_Relative: MC_MoveRelative;
	FB_ReadStatusExtruder: MC_ReadStatus;
	FB_ReadStatusPuller: MC_ReadStatus;
	FB_ResetExtruder: MC_Reset;
	FB_ResetPuller: MC_Reset;
	FB_ManualExtruder: MC_Jog;
	FB_ManualPuller: MC_Jog;
	FB_Power2: MC_Power;
	FB_Power3: MC_Power;
	FB_GearInVelo: MC_GearInVelo;
	FB_GearOut: MC_GearOut;
END_VAR

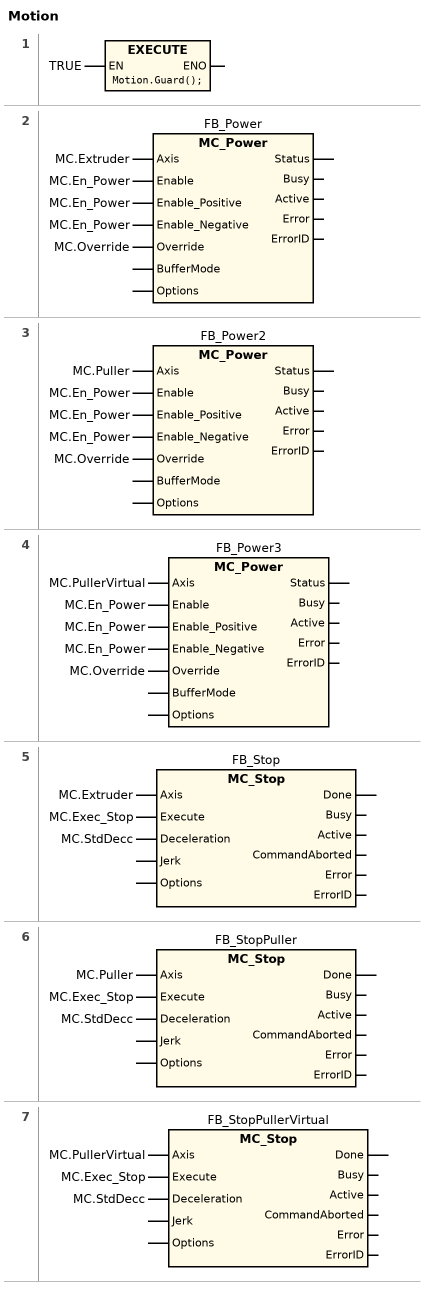
// NETWORK 1
Motion.Guard();

// NETWORK 2
FB_Power(
    Axis := MC.Extruder,
    Enable := MC.En_Power,
    Enable_Positive := MC.En_Power,
    Enable_Negative := MC.En_Power,
    Override := MC.Override); // MC_Power

// NETWORK 3
FB_Power2(
    Axis := MC.Puller,
    Enable := MC.En_Power,
    Enable_Positive := MC.En_Power,
    Enable_Negative := MC.En_Power,
    Override := MC.Override); // MC_Power

// NETWORK 4
FB_Power3(
    Axis := MC.PullerVirtual,
    Enable := MC.En_Power,
    Enable_Positive := MC.En_Power,
    Enable_Negative := MC.En_Power,
    Override := MC.Override); // MC_Power

// NETWORK 5
FB_Stop(Axis := MC.Extruder, Execute := MC.Exec_Stop, Deceleration := MC.StdDecc); // MC_Stop

// NETWORK 6
FB_StopPuller(Axis := MC.Puller, Execute := MC.Exec_Stop, Deceleration := MC.StdDecc); // MC_Stop

// NETWORK 7
FB_StopPullerVirtual(Axis := MC.PullerVirtual, Execute := MC.Exec_Stop, Deceleration := MC.StdDecc); // MC_Stop

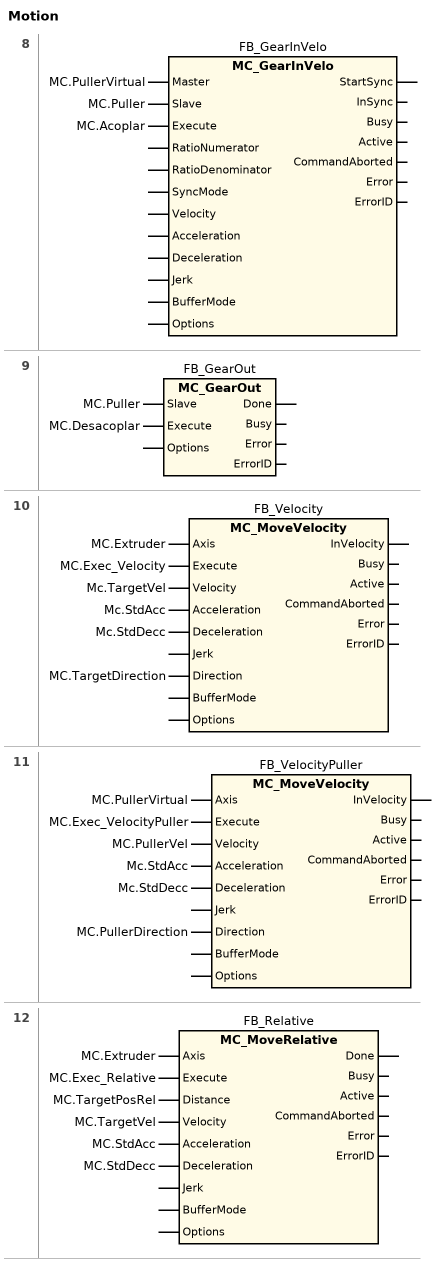
// NETWORK 8
FB_GearInVelo(Master := MC.PullerVirtual, Slave := MC.Puller, Execute := MC.Acoplar); // MC_GearInVelo

// NETWORK 9
FB_GearOut(Slave := MC.Puller, Execute := MC.Desacoplar); // MC_GearOut

// NETWORK 10
FB_Velocity(
    Axis := MC.Extruder,
    Execute := MC.Exec_Velocity,
    Velocity := Mc.TargetVel,
    Acceleration := Mc.StdAcc,
    Deceleration := Mc.StdDecc,
    Direction := MC.TargetDirection); // MC_MoveVelocity

// NETWORK 11
FB_VelocityPuller(
    Axis := MC.PullerVirtual,
    Execute := MC.Exec_VelocityPuller,
    Velocity := MC.PullerVel,
    Acceleration := Mc.StdAcc,
    Deceleration := Mc.StdDecc,
    Direction := MC.PullerDirection); // MC_MoveVelocity

// NETWORK 12
FB_Relative(
    Axis := MC.Extruder,
    Execute := MC.Exec_Relative,
    Distance := MC.TargetPosRel,
    Velocity := MC.TargetVel,
    Acceleration := MC.StdAcc,
    Deceleration := MC.StdDecc); // MC_MoveRelative

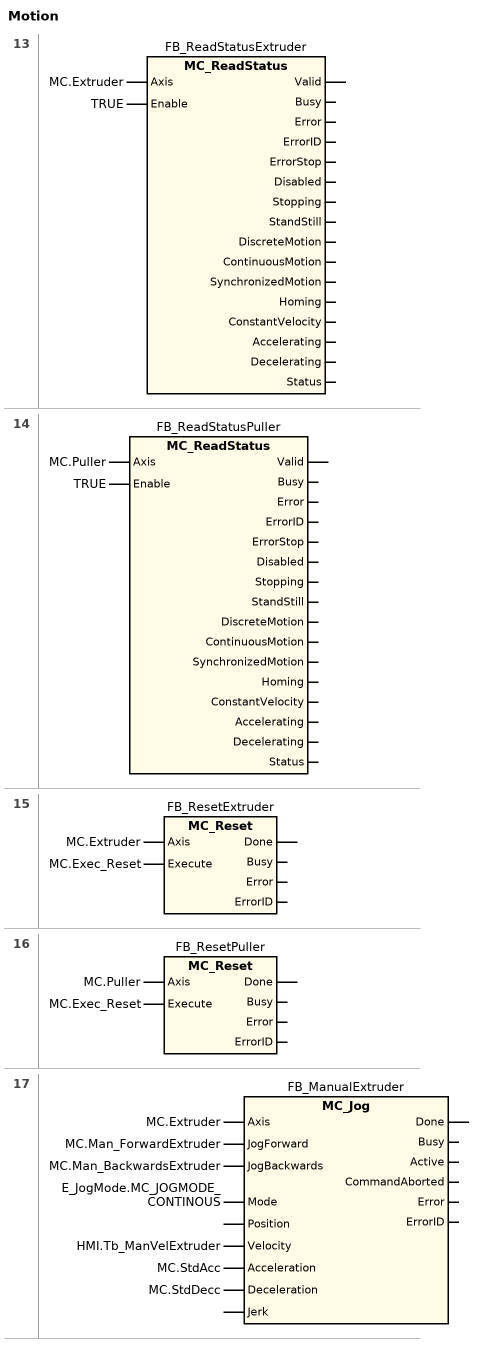
// NETWORK 13
FB_ReadStatusExtruder(Axis := MC.Extruder, Enable := TRUE); // MC_ReadStatus

// NETWORK 14
FB_ReadStatusPuller(Axis := MC.Puller, Enable := TRUE); // MC_ReadStatus

// NETWORK 15
FB_ResetExtruder(Axis := MC.Extruder, Execute := MC.Exec_Reset); // MC_Reset

// NETWORK 16
FB_ResetPuller(Axis := MC.Puller, Execute := MC.Exec_Reset); // MC_Reset

// NETWORK 17
FB_ManualExtruder(
    Axis := MC.Extruder,
    JogForward := MC.Man_ForwardExtruder,
    JogBackwards := MC.Man_BackwardsExtruder,
    Mode := E_JogMode.MC_JOGMODE_CONTINOUS,
    Velocity := HMI.Tb_ManVelExtruder,
    Acceleration := MC.StdAcc,
    Deceleration := MC.StdDecc); // MC_Jog

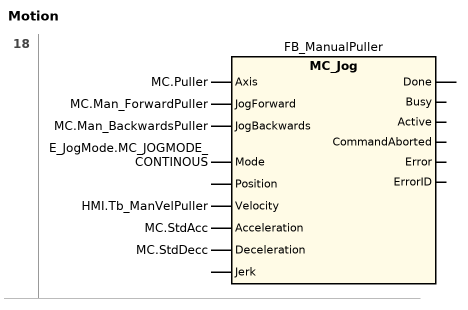
// NETWORK 18
FB_ManualPuller(
    Axis := MC.Puller,
    JogForward := MC.Man_ForwardPuller,
    JogBackwards := MC.Man_BackwardsPuller,
    Mode := E_JogMode.MC_JOGMODE_CONTINOUS,
    Velocity := HMI.Tb_ManVelPuller,
    Acceleration := MC.StdAcc,
    Deceleration := MC.StdDecc); // MC_Jog

ACTION Guard:
MC.Exec_Reset:=FALSE;
IF HMI.Bt_ResetAxis THEN
	IF (MC.Extruder.Status.Error = TRUE) OR (MC.Puller.Status.Error = TRUE) THEN
		MC.Exec_Reset:= TRUE;
	END_IF
END_IF
END_ACTION

ACTION InitMotion:
MC.En_Power := FALSE;
MC.Exec_Relative := FALSE;
MC.Exec_Stop := FALSE;
MC.Exec_Velocity := FALSE;
MC.Exec_VelocityPuller:=FALSE;
MC.Acoplar:=FALSE;
MC.Desacoplar:=FALSE;
IO.Q_VisionLight := FALSE;
END_ACTION

END_PROGRAM

// ---- POUs/ControlTemp.TcPOU
PROGRAM ControlTemp
VAR
	FB_CTRL_TempControllerTop: FB_CTRL_TempController;
	FB_CTRL_TempControllerBot: FB_CTRL_TempController;
	modo:E_CTRL_MODE:=eCTRL_MODE_ACTIVE;
	
	sControllerParameter: ST_CTRL_TempCtrlParameter:=
	(
			(* general parameters *)
			iMode                     :=1,
			bSelCtrlParameterSet      :=TRUE,
			tCtrlCycleTime            :=T#100MS,
			tTaskCycleTime            :=T#10MS,

		  (* tuning parameteer *)
		  iTuningMode               := eCTRL_TuneMode_HEATING,
		  tTuneStabilisation        := T#30S,
		  fEndTunePercentHeating    := 80.0,
		  fYTuneHeating:=100.0,
		  fEndTunePercentCooling    := 20.0,
		  fYStableCooling:=50.0,
		  fScalingFactor            := 1.0,
		
		  (* setpoint parameters *)
		  fWMin:=0.0,
		  fWMax:=573.0,

		  (* start up *)
		  bEnableSoftStart:=FALSE,
		  bEnableRamping:=TRUE,
		  fWStartUp:=348.0,
		  tStartUp:=T#30S,
		  bStartUpRamping:=TRUE,
		  fWStartUpVeloPos:=3.0,
		  fWStartUpVeloNeg:=3.0,
		  fWVeloPos:=5.0,
		  fWVeloNeg:=5.0,
		
		  (* actual value parameters *)
		  bFilter:=FALSE,
		  tFilter:=T#100MS,
		
		  (* deadband parameters *)
		  bDeadband:=FALSE,
		  fEDeadband:=1.0,
		  
		  (* control value parameters *)
		  fYMin:=0.0,
		  fYMax:=573.0,
		  fYManual:=20.0,
		  fYOnFailure:=20.0,
		  tPWMCycleTime:=T#100MS,
		  tPWMMinOffTime:=T#100MS,
		  tPWMMinOnTime:=T#100MS,
		  tPWMWaitingTime:=T#100MS,
		  fYThresholdOff:=50.0,
		  fYThresholdOn:=50.0,
		  nCyclesForSwitchOver      := 100,
		
		  (* controller settings *)
		  bEnablePreController:=FALSE,
		  bEnableZones:=FALSE,
		  bEnableCVFilter:=FALSE,
		  iFilterType:=eCTRL_FilterType_AVERAGE,
		  iControllerType:=eCTRL_ControllerType_PID,
		
		  (* min max temperatures *)
		  TempLow:=283.0,
		  TempLowLow:=0.0,
		  TempHigh:=503.0,
		  TempHighHigh:=523.0,
		  TempAbsoluteHigh:=523.0,
		  TempAbsoluteLow:=0.0,
		
		  (* internal tuning parameters *)
		  fTuneKp                   := 1.2,
		  fTuneTn                   := 2.0,
		  fTuneTv                   := 0.42,
		  fTuneTd                   := 0.25
  );
		
	//sControllerParameter
	sControllerParameter2:ST_CTRL_TempCtrlParameter:=
	(
		(* base *)
		tCtrlCycleTime := T#1000MS,
		tTaskCycleTime := T#10MS,
		
		fYMin := -100,
		fYMax := 100,
		tPWMCycleTime := T#100MS ,
		fYManual := 20,
		bFilter := FALSE,
		tFilter := T#100MS,
		bDeadband := FALSE,
		fEDeadband := 1.0, (* deadband *)
		fWMin := 288,
		fWMax := 523,
		fWStartUp := 323,
		tStartUp := T#1S,
		fWVeloPos := 0.5,
		fWVeloNeg := 0.5,
		bStartUpRamping := TRUE,
		fWStartUpVeloPos := 0.5,
		fWStartUpVeloNeg := 0.5,
		iMode := eCTRL_ControlMode_HEATING,
		dwAlarmSupp := 16#FF_FF_FF_FF,
		bSelCtrlParameterSet:= FALSE,
		
		(* tuninig *)
		iTuningMode := eCTRL_TuneMode_heating,
		fYTuneHeating := 100.0,
		fYTuneCooling := -100.0,
		fEndTunePercentHeating := 80.0, (* switch to closed loop control when X > 0.8*W *)
		fEndTunePercentCooling := -70.0, (* switch to closed loop control when X < 0.2*W *)
		iReactionOnFailure := eCTRL_ReactionOnFailure_StopController,
		TempLow := -50.0,
		TempLowLow := -100.0,
		TempHigh := 523,
		TempHighHigh := 523,
		TempAbsoluteHigh := 523,
		TempAbsoluteLow := -95.0,
		bEnablePreController := FALSE,
		bEnableZones := FALSE,
		bEnableCVFilter := FALSE,
		iFilterType := eCTRL_FilterType_AVERAGE,
		iControllerType := eCTRL_ControllerType_PID
	);
END_VAR

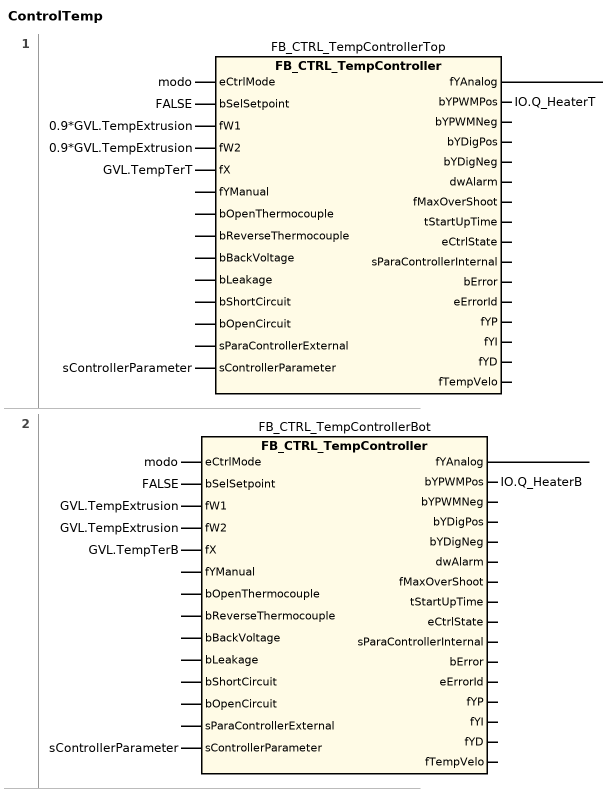
// NETWORK 1
FB_CTRL_TempControllerTop(
    eCtrlMode := modo,
    bSelSetpoint := FALSE,
    fW1 := 0.9*GVL.TempExtrusion,
    fW2 := 0.9*GVL.TempExtrusion,
    fX := GVL.TempTerT,
    sControllerParameter := sControllerParameter,
    bYPWMPos => IO.Q_HeaterT); // FB_CTRL_TempController

// NETWORK 2
FB_CTRL_TempControllerBot(
    eCtrlMode := modo,
    bSelSetpoint := FALSE,
    fW1 := GVL.TempExtrusion,
    fW2 := GVL.TempExtrusion,
    fX := GVL.TempTerB,
    sControllerParameter := sControllerParameter,
    bYPWMPos => IO.Q_HeaterB); // FB_CTRL_TempController

END_PROGRAM

// ---- POUs/GestionVentiladores.TcPOU
PROGRAM GestionVentiladores
VAR
END_VAR

//Inicialmente apaga los ventiladores
IO.Q_Vent1:=0;
IO.Q_Vent2:=0;

IF (GVL.Mode=MODES.AUTO AND MC.Exec_Velocity=TRUE) OR (GVL.Mode=MODES.MAN AND (MC.Man_ForwardExtruder OR MC.Man_BackwardsExtruder)) THEN
	IO.Q_Vent1:=24575; //Alimenta ventilador a 7.5V
	IO.Q_Vent2:=16383;	//Alimenta ventilador a 5V
END_IF

END_PROGRAM

// ---- POUs/MedidaDiamMec.TcPOU
PROGRAM MedidaDiamMec
VAR
	LoopCounter:INT;
	
	//Variables para la lectura de sensores
	MedSenMec:REAL:=0.0;
	MedSensores:REAL:=0.0;
	SumSenOpt: REAL:=0.0;
	MedSenOpt: REAL:=0.0;
	
	//Variables para la media de medidas de los sensores
	Lecturas:ARRAY[0..9] OF REAL:=[10(0.0)]; 	//Medidas del diametro inicializadas
	Index:INT:=0; 								//Indice del vector de medidas 
	Suma:REAL:=0.0; 							//Suma de medidas
	
END_VAR

//Calculo del diametro
MedSenMec:=((IO.I_SMec1+IO.I_SMec2)/2);

//Hacer media de las 10 ultimas medidas del diametro
Suma:= Suma - Lecturas[Index];
Lecturas[index]:=MedSensores;
Suma:=Suma+Lecturas[index];
Index:= Index + 1;
IF (Index > 9) THEN
	Index := 0;    	//Volvemos al inicio del vector
END_IF
GVL.MedidaSensorMecanico:=Suma/10;

END_PROGRAM

// ---- POUs/MedidaTempPuente.TcPOU
PROGRAM MedidaTempPuente
VAR
	VampT:REAL;
	VampB:REAL;
	VAT:REAL;
	VAB:REAL;
	VB:REAL;
	Rpt100T:REAL;
	Rpt100B:REAL;
	TempTerT: INT;
	TempTerB: INT;
	Gain:REAL;
	
	//Variables media de medidas de temperatura
	LecturasT:ARRAY[0..9] OF REAL:=[10(0.0)];
	IndexT:INT:=0; 			//Indice del vector de medidas 
	SumaT:REAL:=0.0; 		//Suma de medidas
	MedidaT:REAL:=0.0; 		//Media de medidas y por tanto medida de la temperatura
	LecturasB:ARRAY[0..9] OF REAL:=[10(0.0)];
	IndexB:INT:=0; 			//Indice del vector de medidas 
	SumaB:REAL:=0.0; 		//Suma de medidas
	MedidaB:REAL:=0.0; 		//Media de medidas y por tanto medida de la temperatura
END_VAR

VAR CONSTANT
	Vcc:REAL:=10.0;
	R1:REAL:=9400;
	//R0:REAL:=100;
	R0:REAL:=101.1;
	Rg:REAL:=983;
	//Gain:REAL:=72.84091;
	//Gain:REAL:=70;
	//Gain:REAL:=101;
	A:LREAL:=3.9083*EXPT(10,-3);
	B:LREAL:=-5.775*EXPT(10,-7);
END_VAR

VB:=(R0*Vcc)/(R1+R0);
Gain:=1.0+(100000.0/Rg);

//Calculo de la temperatura del termico superior
VampT:=((ABS(IO.I_TermTPuente))*Vcc)/32767;

//Hacer media de las 10 ultimas medidas de la temperatura
SumaT:= SumaT - LecturasT[IndexT];
LecturasT[IndexT]:=VampT;
SumaT:=SumaT+LecturasT[IndexT];
IndexT:= IndexT + 1;
IF (IndexT > 9) THEN
	IndexT := 0;    //Volvemos al inicio del vector
END_IF
MedidaT:=SumaT/10;
	
VAT:=(MedidaT/Gain)+VB;
Rpt100T:=(R1)/((Vcc/VAT)-1);
GVL.TempTerT:=(-A+SQRT(A*A-4*B*(1-(Rpt100T/R0))))/(2*B);


//Calculo de la temperatura del termico inferior
VampB:=((ABS(IO.I_TermBPuente))*Vcc)/32767;

//Hacer media de las 10 ultimas medidas de la temperatura
SumaB:= SumaB - LecturasB[IndexB];
LecturasB[IndexB]:=VampB;
SumaB:=SumaB+LecturasB[IndexB];
IndexB:= IndexB + 1;
IF (IndexB > 9) THEN
	IndexB := 0;    //Volvemos al inicio del vector
END_IF
MedidaB:=SumaB/10;

VAB:=(MedidaB/Gain)+VB;
Rpt100B:=(R1)/((Vcc/VAB)-1);
GVL.TempTerB:=(-A+SQRT(A*A-4*B*(1-(Rpt100B/R0))))/(2*B);

END_PROGRAM

// ---- POUs/Database/DatabaseManager.TcPOU
FUNCTION_BLOCK PUBLIC DatabaseManager
VAR_INPUT
	Execute:BOOL;
	SQLCmd:STRING[999];
END_VAR

VAR_IN_OUT
	
END_VAR
	
VAR_OUTPUT
	rec:POINTER TO BYTE;
END_VAR
VAR
	bCONNECT: BOOL;
	bEXECUTE: BOOL;
	bREAD : BOOL;
	bDISCONNECT: BOOL;
	R_TRIG1: R_TRIG;
	R_TRIG2: R_TRIG;
	R_TRIG3: R_TRIG;
	R_TRIG4: R_TRIG;
	nState: INT;
	nState_Connect: INT;
	nState_Disconnect: INT;
	bConn: BOOL;
	bSP: BOOL;
	bResult: BOOL;
	bData: BOOL;
	nDBID: UDINT := 1;
	fbSQLDatabase: FB_SQLDatabaseEvt(sNetID:='', tTimeout:=T#10S);
	fbSQLStoredProcedure: FB_SQLStoredProcedureEvt(sNetID:='', tTimeout:=T#10S);
	fbSQLResult: FB_SQLResultEvt(sNetID:='', tTimeout:=T#10S);
	
	fbSQLCommandEvt: FB_SQLCommandEvt(sNetId:='',tTimeout:=T#10S);
	
	Cmd:STRING[500]:='SELECT CONVERT(VARBINARY(16), ID) AS [ByteArray], [Name], [Description], [BedTemperature], [HotendTemperature], [IdealTempExtr], [MinTempExtr], [MaxTempExtr] FROM [dbo].[Material] ';
	arrParameter: ARRAY [0..0] OF ST_SQLSPParameter;
	nCustomerID: DINT := 12345;
	nRecordStartIndex: UDINT;
	stRecordArr: ARRAY [1..20] OF ST_Material;
	nRecs: UDINT;
	bError : BOOL;
	nEventID: UDINT;
	sEventClass : STRING(255);
	sEventMsg : STRING(255);
END_VAR

R_TRIG1(CLK:=bCONNECT);
IF R_TRIG1.Q AND nState = 0 THEN
	nState := 1;
END_IF
R_TRIG2(CLK:=bEXECUTE);
IF R_TRIG2.Q AND nState = 0 THEN
	nState := 2;
END_IF
R_TRIG3(CLK:=bREAD);
IF R_TRIG3.Q AND nState = 0 THEN
	nState := 3;
END_IF
R_TRIG4(CLK:=bDISCONNECT);
IF R_TRIG4.Q THEN
	nState := 4;
END_IF

CASE nState OF
0:(*Idle*)
;
1: // Connect to database and create stored procedure instance
	CASE nState_Connect OF
	0:
		IF fbSQLDatabase.Connect(hDBID:= nDBID) THEN
			bConn := NOT fbSQLDatabase.bError;
			IF bConn THEN
				nState_Connect := 1;
			ELSE
				nState:=200;
			END_IF
		END_IF
	1:
		arrParameter[0].sParameterName := '@Customer_ID';
		arrParameter[0].eParameterDataType :=
		Tc3_Database.E_ColumnType.Integer;
		arrParameter[0].eParameterType := E_SPParameterType.Input;
		arrParameter[0].nParameterSize := SIZEOF(nCustomerID);
		IF fbSQLDatabase.CreateCmd(ADR(fbSQLCommandEvt)) THEN
			bSP := NOT fbSQLDatabase.bError;
			nState_Connect:=0;
			nState := 200;
		END_IF
	END_CASE
2: // Execute command
	IF fbSQLCommandEvt.ExecuteDataReturn(pSQLCmd:= ADR(Cmd),cbSQLCmd:= SIZEOF(Cmd),pSQLDBResult:= ADR(fbSQLResult)) THEN
		MEMSET(ADR(stRecordArr),0,SIZEOF(stRecordArr));
		bResult := NOT fbSQLStoredProcedure.bError;
		nState := 200;
	END_IF
3: // Read customer positions
	IF fbSQLResult.Read(nRecordStartIndex, 20, ADR(stRecordArr),SIZEOF(stRecordArr), TRUE, FALSE) THEN
		bData := NOT fbSQLStoredProcedure.bError;
		nRecs := fbSQLResult.nDataCount;
		nState := 200;
	END_IF
4:// Disconnect all
	CASE nState_Disconnect OF
	0:
		IF bData THEN
			IF fbSQLResult.Release() THEN
				nState_Disconnect := 1;
			END_IF
		ELSE
			nState_Disconnect := 1;
		END_IF
	1:
		IF bSP THEN
			IF fbSQLDatabase.Disconnect()THEN
				nState_Disconnect := 2;
			END_IF
		ELSE
			nState_Disconnect := 2;
		END_IF
	2:
		bData := FALSE;
		bSP := FALSE;
		bConn := FALSE;
		bResult := FALSE;
		nEventID := 0;
		bError := FALSE;
		nState_Disconnect := 0;
		nState := 0;
	END_CASE
END_CASE

END_FUNCTION_BLOCK

// ---- POUs/MAIN.TcPOU
PROGRAM MAIN
VAR
	En:BOOL;
	Shot:BOOL;
	Result:ARRAY [0..7] OF REAL;
END_VAR

Motion.InitMotion();
GVL.Vision();

//Medida temperatura
//MedidaTempPuente();	//Medir la temperatura de los termicos con el puente de resistencias
MedidaTempTarjeta();	//Medir la temperatura de los termicos con la tarjeta EL3202

//ControlTemp();		//Gestion temperatura con bloques TF4110

MedidaDiamMec();	//Medida del diametro con el sensor mecanico

OperatingModes();

IF GVL.Mode = Modes.AUTO THEN
	Basic();
END_IF

Manual();
VisuLogic();
Motion();
GestionVentiladores();

END_PROGRAM

// ---- POUs/MedidaTempTarjeta.TcPOU
PROGRAM MedidaTempTarjeta
VAR
END_VAR

GVL.TempTerB:=IO.I_TermB/10.0;

GVL.TempTerT:=IO.I_TermT/10.0;

END_PROGRAM

// ---- POUs/OperatingModes.TcPOU
PROGRAM OperatingModes
VAR
	AuxStopping:Modes;
END_VAR

CASE GVL.Mode OF
	
	// Emergency stop
	Modes.STOP_EM:
		IF HMI.Bt_Rearm THEN
			gvl.Mode := modes.STOP_OP;
		END_IF
	
	// Operative stop
	Modes.STOP_OP:
		IF HMI.Bt_EmStop THEN
			GVL.Mode := Modes.STOP_EM;
		END_IF
		IF HMI.Bt_Run AND HMI.S_ManAuto THEN
			GVL.Mode := Modes.AUTO;
			GVL.State:=0;
		END_IF
		IF NOT HMI.S_ManAuto THEN
			GVL.Mode := Modes.MAN;
		END_IF
		
	// Automatic
	Modes.AUTO:
		IF HMI.Bt_EmStop THEN
			GVL.Mode := Modes.STOP_EM;
		END_IF
		IF NOT HMI.S_ManAuto THEN
			GVL.Mode := Modes.MAN;
		END_IF
		IF HMI.Bt_Stop THEN
			GVL.Mode := Modes.Stopping;
			AuxStopping := Modes.STOP_OP;
		END_IF
		
	// Manual
	Modes.MAN:
		IF HMI.Bt_EmStop THEN
			GVL.Mode := Modes.STOP_EM;
		END_IF
		IF HMi.S_ManAuto THEN
			GVL.Mode := Modes.STOP_OP;
		END_IF	
		
	// Stopping
	Modes.Stopping:
		MC.Exec_Stop:= TRUE;
		IF (Motion.FB_Stop.Done AND Motion.FB_StopPuller.Done AND Motion.FB_StopPullerVirtual.Done AND Motion.FB_GearOut.Done) OR MC.Extruder.Status.Error OR MC.Puller.Status.Error OR MC.PullerVirtual.Status.Error THEN
			GVL.Mode := AuxStopping;
		END_IF
END_CASE

// Axis Power when not in stop
IF GVL.Mode = Modes.AUTO OR GVL.Mode = Modes.Stopping THEN
	MC.En_Power := TRUE;
END_IF

END_PROGRAM

// ---- POUs/Operation/Basic.TcPOU
PROGRAM Basic
VAR
	LoopCounter:INT; //Para pasar de pixeles a mm en el vector de resultados	

	//Variables para la lectura de sensores
	MedSensores:REAL:=0.0;
	SumSenOpt: REAL:=0.0;
	MedSenOpt: REAL:=0.0;
	
	//Variables para la media de medidas de los sensores
	Lecturas:ARRAY[0..9] OF REAL:=[10(0.0)]; 	//Medidas del diametro inicializadas
	Index:INT:=0; 								//Indice del vector de medidas 
	Suma:REAL:=0.0; 							//Suma de medidas
	Medida:REAL:=0.0; 							//Media de medidas y por tanto medida del diametro
END_VAR

//STATE CONTROL
CASE GVL.State OF
	0:  IF HMI.Bt_StartCycle THEN 	//Se pulsa start
			GVL.State:=1;
	END_IF
	IF HMI.Bt_StopCycle THEN 		//Se pulsa stop
		GVL.State:=30;
	END_IF
	
	1:  IF Motion.FB_Power.Status AND Motion.FB_Power2.Status AND Motion.FB_Power3.Status THEN 	//Estan motores en potencia
			GVL.State:=2;
	END_IF
	IF HMI.Bt_StopCycle THEN 		//Se pulsa stop
		GVL.State:=30;
	END_IF
	
	2: IF (GVL.TempTerB>=HMI.Tb_Temp) AND (GVL.TempTerT>=(0.95*HMI.Tb_Temp)) THEN 				//En temperatura
			GVL.State:=3;
	END_IF
	IF HMI.Bt_StopCycle THEN 		//Se pulsa stop
		GVL.State:=30;
	END_IF
	
	3: IF Motion.FB_VelocityPuller.InVelocity AND Motion.FB_Velocity.InVelocity THEN 			//Eje de extrusora y virtual del puller a la velocidad indicada
		GVL.State:=4;
	END_IF
	IF HMI.Bt_StopCycle THEN 		//Se pulsa stop
			GVL.State:=30;
	END_IF
	
	4: IF Motion.FB_GearInVelo.InSync THEN 	//Ejes acoplados
		GVL.State:=5;
	END_IF
	IF HMI.Bt_StopCycle THEN 		//Se pulsa stop
			GVL.State:=30;
	END_IF
	
	5: IF GVL.NuevaMedidaCamara THEN 	//Nueva foto de la camara
		GVL.State:=6;
		// Restablecer valores de medida para una futura medida
		GVL.NuevaMedidaCamara:=FALSE;
		GVL.Vision.SingleShot(Enable:=TRUE, Execute:=FALSE);
	END_IF
	IF HMI.Bt_StopCycle THEN 		//Se pulsa stop
			GVL.State:=30;
	END_IF
	
	6: 
	IF HMI.Bt_StopCycle THEN 		//Se pulsa stop
			GVL.State:=30;
	END_IF
	
	7: GVL.State:=5;
	IF HMI.Bt_StopCycle THEN 		//Se pulsa stop
			GVL.State:=30;
	END_IF
	
	30: IF (Motion.FB_Stop.Done AND Motion.FB_StopPuller.Done AND Motion.FB_StopPullerVirtual.Done AND Motion.FB_GearOut.Done) THEN 	//Ejes parados y desacoplados
		GVL.State:=0;
	END_IF
END_CASE

//ACT
CASE GVL.State OF
	
	2: IO.Q_HeaterB:=TRUE;
	IO.Q_HeaterT:=TRUE;
	
	3: 
	//Extruder
	MC.TargetDirection:= MC_Direction.MC_Positive_Direction;
	MC.TargetVel:= HMI.Tb_Vel;
	MC.Exec_Velocity:=TRUE;
	//Puller
	MC.PullerDirection:= MC_Direction.MC_Positive_Direction;
	MC.PullerVel:=GVL.ActPuller;
	MC.Exec_VelocityPuller:=TRUE;
	//Vision
	IO.Q_VisionLight := TRUE;
	
	4: MC.Acoplar:=TRUE;
	//Puller
	MC.Exec_VelocityPuller:=TRUE;
	//Vision
	IO.Q_VisionLight := TRUE;
	
	5: 
	//Puller
	MC.Exec_VelocityPuller:=TRUE;
	//Vision
	IO.Q_VisionLight := TRUE;
	
	6:
	//Puller
	MC.Exec_VelocityPuller:=TRUE;
	//Vision
	IO.Q_VisionLight := TRUE;
	
	7: MC.PullerVel:=GVL.ActPuller;
	//Vision
	IO.Q_VisionLight := TRUE;
	
	30: MC.Desacoplar:=TRUE;
	MC.Exec_Stop:=TRUE;
END_CASE

IF (GVL.State=1) THEN 	//Comprobacion de la variable de configuracion, el diametro de trabajo y con el la velocidad inicial del puller
	IF GVL.config THEN
		GVL.dReferencia:=2.85;
		GVL.ActPuller:=(360/125.6637)*(6.43025*HMI.Tb_Vel)/(GVL.dReferencia*GVL.dReferencia);
	ELSE
		GVL.dReferencia:=1.75;
		GVL.ActPuller:=(360/125.6637)*(6.43025*HMI.Tb_Vel)/(GVL.dReferencia*GVL.dReferencia);
	END_IF
END_IF

IF (GVL.State=5) THEN //Proceso de nueva foto y gestion de los termicos
	
	//Gestion de temperatura para extrusion. PLA: TB_Temp=200ºC (rango de 198-210ºC debido a tiempo de medida del Pt100)
	IF (GVL.TempTerT>(HMI.Tb_Temp*0.95)) THEN 	//Gestiona el calentador superior
		IO.Q_HeaterT:=FALSE;
	END_IF
	IF (GVL.TempTerT<(HMI.Tb_Temp*0.95-1.0)) THEN
		IO.Q_HeaterT:=TRUE;
	END_IF
	
	IF (GVL.TempTerB>(HMI.Tb_Temp)) THEN 		//Gestiona el calentador inferior
		IO.Q_HeaterB:=FALSE;
	END_IF
	IF (GVL.TempTerB<(HMI.Tb_Temp-1.0)) THEN
		IO.Q_HeaterB:=TRUE;
	END_IF
	
	//Medida con la camara del diametro del filamento
	GVL.Vision.SingleShot(Enable:=TRUE, 
					Execute:=TRUE,
					Q=>GVL.VisionResults,
					Measurement=>GVL.NuevaMedidaCamara);
END_IF

IF (GVL.State=6) THEN 	//Nueva medida de la camara. Calculo del diametro medido con los sensores y calculo de actuacion del puller
	SumSenOpt:=0.0;
	FOR LoopCounter:=0 TO 7 BY 1 DO
		GVL.VisionResultsmm[LoopCounter] := GVL.VisionResults[LoopCounter]*GVL.ScalingFactor;
		SumSenOpt:=GVL.VisionResultsmm[LoopCounter]+SumSenOpt;
	END_FOR	
	MedSenOpt:=SumSenOpt/3;
		
	//Calculo del diametro
	MedSensores:=((GVL.MedidaSensorMecanico+MedSenOpt)/2);
		
	//Hacer media de las 10 ultimas medidas del diametro
	Suma:= Suma - Lecturas[Index];
	Lecturas[index]:=MedSensores;
	Suma:=Suma+Lecturas[index];
	Index:= Index + 1;
	IF (Index > 9) THEN
		Index := 0;    	//Volvemos al inicio del vector
	END_IF
	Medida:=Suma/10;
		
	//Gestion de la actuacion
	IF (Medida>(GVL.dReferencia+GVL.dTolerancia)) THEN 		//Diametro grande
		GVL.ActPuller:=GVL.ActPuller+GVL.vPaso;
		GVL.State:=7;
	END_IF
	
	IF (Medida<(GVL.dReferencia-GVL.dTolerancia)) THEN 		//Diametro pequeño
		GVL.ActPuller:=GVL.ActPuller-GVL.vPaso;
		GVL.State:=7;
	END_IF
	
	IF (Medida<(GVL.dReferencia+GVL.dTolerancia)) AND (Medida>(GVL.dReferencia-GVL.dTolerancia)) THEN 	//Diametro correcto
		GVL.State:=5;
	END_IF
	
	//Limitador de la actuacion
	IF (GVL.ActPuller>GVL.ActPuller_Max) THEN 
		GVL.ActPuller:=GVL.ActPuller_Max;
	ELSIF (GVL.ActPuller<GVL.ActPuller_Min) THEN
		GVL.ActPuller:=GVL.ActPuller_Min;
	END_IF
		
END_IF

END_PROGRAM

// ---- POUs/VISUCode/VisuLogic.TcPOU
PROGRAM VisuLogic
VAR_OUTPUT
	L_Run: BOOL;
	L_StopOP: BOOL;
	L_StopEM: BOOL;
	L_Manual: BOOL;
	
	
END_VAR
VAR
	T_StopOP: TON;
	Time_Stop: TIME := T#1S;
END_VAR


L_Run := (GVL.Mode = Modes.AUTO);
L_Manual := (GVL.Mode = Modes.MAN);
L_StopEM := (GVL.Mode = Modes.STOP_EM);
IF GVL.Mode <> Modes.STOP_OP THEN
	L_stopOP := FALSE;
END_IF

//Timing Stop OP
IF GVL.Mode = Modes.STOP_OP THEN
	T_StopOP(IN:=TRUE, PT:=Time_Stop);
	IF T_StopOP.Q THEN
		T_StopOP(IN:=FALSE);
		L_StopOP := NOT L_StopOP;
	END_IF
END_IF

END_PROGRAM

// ---- GlobalTextList.TcGTLO
TEXTLIST GlobalTextList
  456 = '%.2f'
  791 = '%.2f ºC'
  406 = '%.3f'
  446 = '%.4F'
  479 = '%.4f'
  377 = '%.4f mm'
  56 = '%.4f px'
  403 = '%s'
  734 = '%s ºC'
  892 = 'Activate'
  111 = 'Activate\nContinuous' | Galician: 'Activar\ncontinuo' | Español: 'Activar\ncontinuo'
  419 = 'Activate\nSingle' | Galician: 'Activar\núnico'
  600 = 'Auto             Manual'
  864 = 'Auto        Manual'
  794 = 'Automatic' | Galician: 'Automático'
  270 = 'Backwards'
  279 = 'Basic Mode' | Galician: 'Modo básico'
  809 = 'Bottom\nHeater' | Galician: 'Calefactor\ninferior'
  481 = 'Bottom Heater' | Galician: 'Calefactor inferior'
  131 = 'BUSY'
  922 = 'Camera' | Galician: 'Cámara'
  766 = 'Emergency' | Galician: 'Emerxencia'
  497 = 'ERR'
  130 = 'Error' | Galician: 'Erro'
  673 = 'Extruder' | Galician: 'Extrusor'
  543 = 'Extruder Motion'
  887 = 'FLC'
  296 = 'FLG'
  32 = 'Forward'
  6 = 'GroupBox'
  358 = 'Heater Group'
  461 = 'Light'
  542 = 'Manual' | Galician: 'Manual'
  277 = 'Mediciones de la cámara' | Galician: 'Medicións da camara'
  963 = 'Medida1'
  722 = 'Medida2'
  161 = 'Medida3'
  420 = 'Medida4'
  375 = 'Medida5'
  65 = 'Medida6'
  644 = 'Medida7'
  316 = 'Medida8'
  668 = 'Modo: %s'
  151 = 'Motion'
  653 = 'Moving' | Galician: 'Movendose'
  808 = 'NEW'
  548 = 'NG'
  275 = 'Operating modes' | Galician: 'Modos de operación'
  139 = 'Power' | Galician: 'Potencia'
  650 = 'Puller Motion'
  586 = 'Rearm' | Galician: 'Rearme'
  989 = 'Shoot'
  280 = 'Shot' | Galician: 'Capturar'
  688 = 'Start' | Galician: 'Inicio'
  765 = 'Start Cycle' | Galician: 'Iniciar ciclo'
  869 = 'State' | Galician: 'Estado'
  988 = 'Status' | Galician: 'Estado'
  954 = 'Stop' | Galician: 'Parada'
  385 = 'STOP' | Galician: 'Paro'
  835 = 'Stop Cycle' | Galician: 'Parar Ciclo'
  25 = 'Temperatura calentamiento (ºC): %s'
  524 = 'Temperature' | Galician: 'Temperatura'
  386 = 'Termal Group'
  847 = 'Top' | Galician: 'Superior'
  503 = 'Top\nHeater' | Galician: 'Calefactor\nsuperior'
  559 = 'Top Heater' | Galician: 'Calefactor superior'
  81 = 'Velocidad extrusora (deg/s): %s'
  367 = 'Velocity' | Galician: 'Velocidade'
  843 = 'Velocity (deg/s)'
END_TEXTLIST

// ---- VISUs/BasicHMI.TcVIS
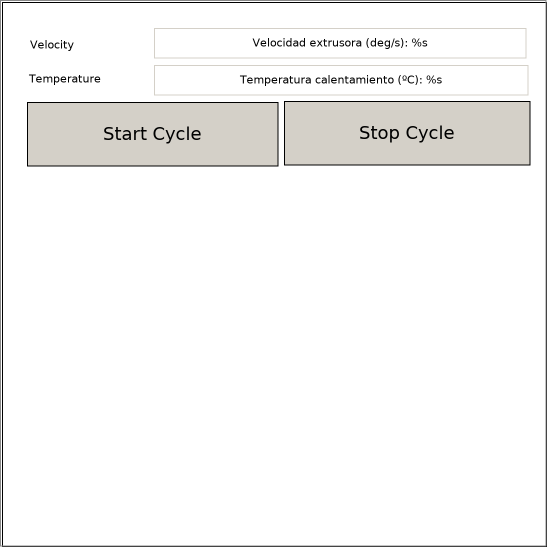
VISUALIZATION BasicHMI  // 547x547
    Rectangle (2,2 545x545)
    Textfield (154,28 372x30), "Velocidad extrusora (deg/s): %s", text variable: HMI.Tb_Vel
        OnMouseDown: write HMI.Tb_Vel via VisuDialogs.Numpad
    Label (27,30 120x30), "Velocity"
    Rectangle (27,102 251x64), "Start Cycle"
        tap HMI.Bt_StartCycle
    Label (26,64 120x30), "Temperature"
    Textfield (154,65 374x30), "Temperatura calentamiento (ºC): %s", text variable: HMI.Tb_Temp
        OnMouseDown: write HMI.Tb_Temp via VisuDialogs.Keypad
    Rectangle (284,101 246x64), "Stop Cycle"
        tap HMI.Bt_StopCycle
END_VISUALIZATION

// ---- VISUs/MainHMI.TcVIS
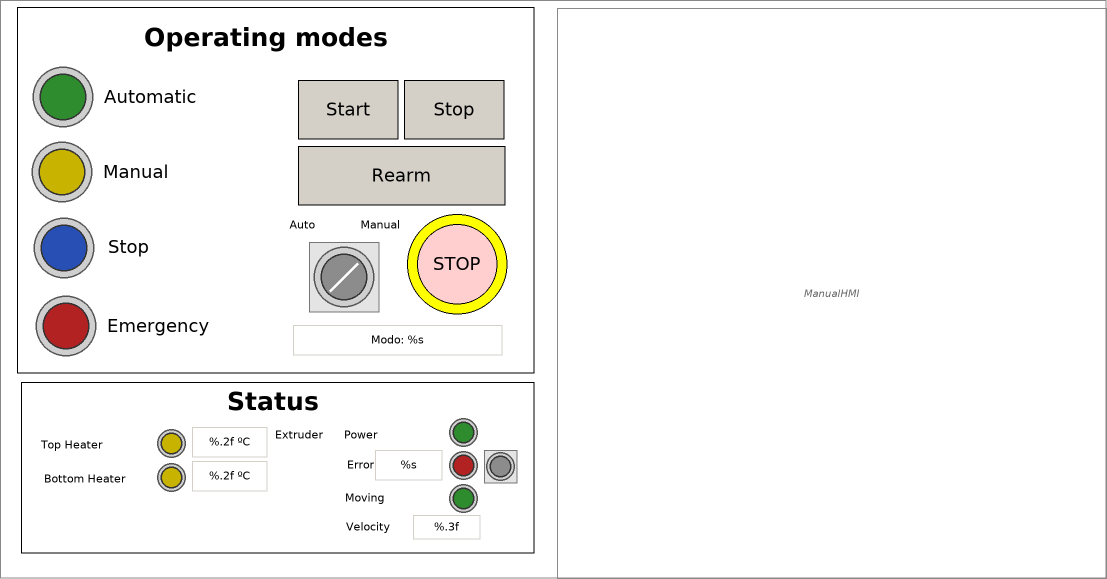
VISUALIZATION MainHMI  // 1107x579
    RoundedRectangle (21,382 513x171)
    RoundedRectangle (17,7 517x366)
    Lamp1 (28,62 70x70), variable: VisuLogic.L_Run, style: Lamp-Lamp1-Green
    Label (101,82 118x30), "Automatic"
    Label (100,157 119x30), "Manual"
    Lamp1 (27,137 70x70), variable: VisuLogic.L_Manual, style: Lamp-Lamp1-Yellow
    Label (105,232 114x30), "Stop"
    Lamp1 (29,213 70x70), variable: VisuLogic.L_StopOP, style: Lamp-Lamp1-Blue
    Label (104,311 115x30), "Emergency"
    Lamp1 (31,291 70x70), variable: VisuLogic.L_StopEM, style: Lamp-Lamp1-Red
    Rectangle (298,80 100x59), "Start"
        tap HMI.Bt_Run
    Rectangle (404,80 100x59), "Stop"
        tap HMI.Bt_Stop
    Rectangle (298,146 207x59), "Rearm"
        tap HMI.Bt_Rearm
    Ellipse (407,214 100x100)
    Ellipse (417,224 80x80), "STOP"
        toggle HMI.Bt_EmStop
    RotarySwitch (309,242 70x70), variable: HMI.S_ManAuto, behaviour: TOGGLE, style: Switch-RotarySwitch-Gray
    Label (284,210 122x30), "Auto Manual"
    Label (124,22 284x30), "Operating modes"
    Label (131,386 284x30), "Status"
    Lamp1 (155,427 33x33), variable: IO.Q_HeaterT, style: Lamp-Lamp1-Yellow
    Lamp1 (155,461 33x33), variable: IO.Q_HeaterB, style: Lamp-Lamp1-Yellow
    Label (38,430 150x30), "Top Heater"
    Label (41,464 150x30), "Bottom Heater"
    Textfield (192,427 75x30), "%.2f ºC", text variable: GVL.TempTerT
    Textfield (192,461 75x30), "%.2f ºC", text variable: GVL.TempTerB
    Label (272,420 57x30), "Extruder"
    Lamp1 (447,449 33x33), variable: MC.Extruder.Status.Error, style: Lamp-Lamp1-Red
    Lamp1 (447,416 33x33), variable: Motion.FB_Power.Status, style: Lamp-Lamp1-Green
    Label (341,420 57x30), "Power"
    Label (344,450 57x30), "Error"
    Textfield (375,450 67x30), "%s", text variable: MC.Extruder.Status.ErrorID
    Lamp1 (447,482 33x33), variable: MC.Extruder.Status.Moving, style: Lamp-Lamp1-Green
    Label (342,483 103x30), "Moving"
    Label (343,512 57x30), "Velocity"
    Textfield (413,515 67x24), "%.3f", text variable: MC.Extruder.NcToPlc.ActVelo
    Textfield (293,325 209x30), "Modo: %s", text variable: GVL.Mode
    PushSwitch (484,450 33x33), variable: HMI.Bt_ResetAxis, behaviour: TAP, style: Switch-PushSwitch-Gray
    TabControl (557,8 550x571)
        shows ManualHMI()
        shows VisionHMI()
        shows BasicHMI()
        [0]: TabTitle=Manual
        [1]: TabTitle=Camera
        [2]: TabTitle=Basic Mode
END_VISUALIZATION

// ---- VISUs/ManualHMI.TcVIS
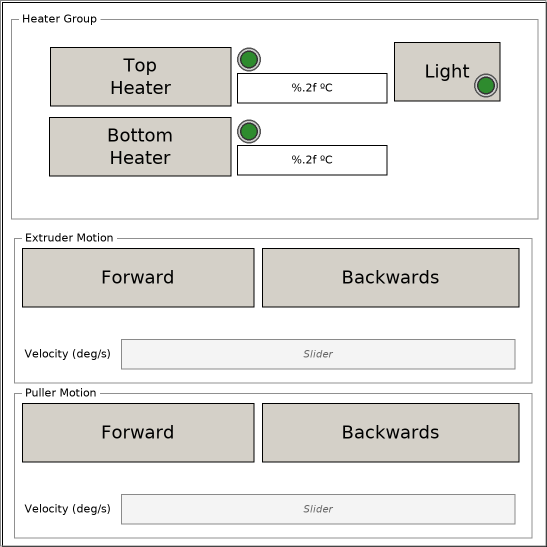
VISUALIZATION ManualHMI  // 547x547
    Rectangle (2,2 545x545)
    GroupBox (11,11 527x208), "Heater Group"
        Rectangle (39,36 181x59), "Top Heater"
            toggle HMI.Bt_ManHeatTop
        Rectangle (226,62 150x30), "%.2f ºC", text variable: GVL.TempTerT
        Rectangle (226,134 150x30), "%.2f ºC", text variable: GVL.TempTerB
        Lamp1 (224,107 28x27), variable: IO.Q_HeaterB, style: Lamp-Lamp1-Green
        Lamp1 (224,35 28x27), variable: IO.Q_HeaterT, style: Lamp-Lamp1-Green
        Rectangle (38,106 182x59), "Bottom Heater"
            toggle HMI.Bt_ManHeatBot
        Rectangle (383,31 106x59), "Light"
            toggle HMI.Bt_Light
        Lamp1 (461,61 28x27), variable: IO.Q_VisionLight, style: Lamp-Lamp1-Green
    GroupBox (14,230 518x153), "Extruder Motion"
        Rectangle (8,18 232x59), "Forward"
            tap HMI.Bt_ManForwardExtruder
        Rectangle (248,18 257x59), "Backwards"
            tap HMI.Bt_ManBackwardsExtruder
        Slider (107,109 394x30), variable: HMI.Tb_ManVelExtruder, scale 0..720
        Label (2,109 104x30), "Velocity (deg/s)"
    GroupBox (14,385 518x153), "Puller Motion"
        Rectangle (8,18 232x59), "Forward"
            tap HMI.Bt_ManForwardPuller
        Rectangle (248,18 257x59), "Backwards"
            tap HMI.Bt_ManBackwardsPuller
        Slider (107,109 394x30), variable: HMI.Tb_ManVelPuller, scale 0..720
        Label (2,109 104x30), "Velocity (deg/s)"
END_VISUALIZATION

// ---- VISUs/VisionHMI.TcVIS
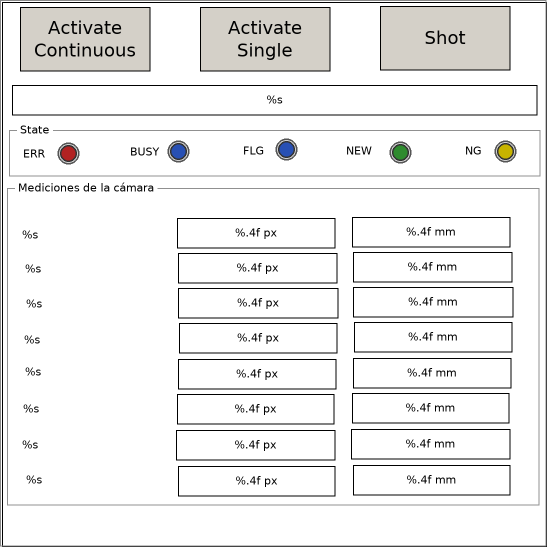
VISUALIZATION VisionHMI  // 547x547
    Rectangle (2,2 545x545)
    Rectangle (200,7 130x64), "Activate Single"
        toggle HMI.Bt_ActivateSingle
    Rectangle (12,85 525x30), "%s", text variable: GVL.Vision.State
    Rectangle (380,6 130x64), "Shot"
        tap HMI.Bt_Shot
    GroupBox (7,180 532x325), "Mediciones de la cámara"
        Rectangle (170,38 158x30), "%.4f px", text variable: GVL.VisionResults[0]
        Rectangle (171,73 159x30), "%.4f px", text variable: GVL.VisionResults[1]
        Rectangle (171,108 160x30), "%.4f px", text variable: GVL.VisionResults[2]
        Rectangle (172,143 158x30), "%.4f px", text variable: GVL.VisionResults[3]
        Rectangle (171,179 158x30), "%.4f px", text variable: GVL.VisionResults[4]
        Rectangle (170,214 157x30), "%.4f px", text variable: GVL.VisionResults[5]
        Rectangle (169,250 159x30), "%.4f px", text variable: GVL.VisionResults[6]
        Rectangle (171,286 157x30), "%.4f px", text variable: GVL.VisionResults[7]
        Rectangle (345,37 158x30), "%.4f mm", text variable: GVL.VisionResultsmm[0]
        Rectangle (12,40 150x30), "%s", text variable: HMI.MeasurementNames[0]
        Rectangle (15,74 150x30), "%s", text variable: HMI.MeasurementNames[1]
        Rectangle (16,109 150x30), "%s", text variable: HMI.MeasurementNames[2]
        Rectangle (14,145 150x30), "%s", text variable: HMI.MeasurementNames[3]
        Rectangle (15,177 150x30), "%s", text variable: HMI.MeasurementNames[4]
        Rectangle (13,214 150x30), "%s", text variable: HMI.MeasurementNames[5]
        Rectangle (12,250 150x30), "%s", text variable: HMI.MeasurementNames[6]
        Rectangle (16,285 150x30), "%s", text variable: HMI.MeasurementNames[7]
    Rectangle (20,7 130x64), "Activate Continuous"
        toggle HMI.Bt_ActivateContinuous
    GroupBox (9,122 531x54), "State"
        Label (11,17 32x30), "ERR"
        Lamp1 (45,19 29x25), variable: GVL.Vision.SensorToPlc.ERR, style: Lamp-Lamp1-Red
        Label (118,15 38x30), "BUSY"
        Lamp1 (155,17 29x25), variable: GVL.Vision.SensorToPlc.BUSY, style: Lamp-Lamp1-Blue
        Label (231,14 38x30), "FLG"
        Lamp1 (263,15 29x25), variable: GVL.Vision.SensorToPlc.FLG, style: Lamp-Lamp1-Blue
        Label (334,14 38x30), "NEW"
        Lamp1 (377,18 29x25), variable: GVL.NuevaMedidaCamara, style: Lamp-Lamp1-Green
        Label (453,14 38x30), "NG"
        Lamp1 (482,17 29x25), variable: GVL.Vision.SensorToPlc.OR_Jud, style: Lamp-Lamp1-Yellow
    Rectangle (353,252 159x30), "%.4f mm", text variable: GVL.VisionResultsmm[1]
    Rectangle (353,287 160x30), "%.4f mm", text variable: GVL.VisionResultsmm[2]
    Rectangle (354,322 158x30), "%.4f mm", text variable: GVL.VisionResultsmm[3]
    Rectangle (353,358 158x30), "%.4f mm", text variable: GVL.VisionResultsmm[4]
    Rectangle (352,393 157x30), "%.4f mm", text variable: GVL.VisionResultsmm[5]
    Rectangle (351,429 159x30), "%.4f mm", text variable: GVL.VisionResultsmm[6]
    Rectangle (353,465 157x30), "%.4f mm", text variable: GVL.VisionResultsmm[7]
END_VISUALIZATION
